// Check for changes (uncomment/comment to choose which values should be compared!)
IF ( (iVehicleID >= 1) AND (iVehicleID <= MM_MAX_NUMBER_OF_VEHICLE_ELEMENTS) ) THEN
	IF ( 	(aReadVehicleData[iVehicleID].stVehicle.bDataValid <> aOldVehicleData[iVehicleID].bDataValid) OR
			(aReadVehicleData[iVehicleID].stVehicle.bMaterial <> aOldVehicleData[iVehicleID].bMaterial) OR
			(aReadVehicleData[iVehicleID].stVehicle.bNOK <> aOldVehicleData[iVehicleID].bNOK) OR
			(aReadVehicleData[iVehicleID].stVehicle.bTool <> aOldVehicleData[iVehicleID].bTool) OR
			(aReadVehicleData[iVehicleID].stVehicle.bVehiclePresent <> aOldVehicleData[iVehicleID].bVehiclePresent) OR
//			(aReadVehicleData[iVehicleID].stVehicle.fPosition <> aOldVehicleData[iVehicleID].fPosition) OR
//			(aReadVehicleData[iVehicleID].stVehicle.fTargetPosition <> aOldVehicleData[iVehicleID].fTargetPosition) OR
//			(aReadVehicleData[iVehicleID].stVehicle.fVelocity <> aOldVehicleData[iVehicleID].fVelocity) OR
//			(aReadVehicleData[iVehicleID].stVehicle.nPathID <> aOldVehicleData[iVehicleID].nPathID) OR
			(aReadVehicleData[iVehicleID].stVehicle.nPriority <> aOldVehicleData[iVehicleID].nPriority) OR
//			(aReadVehicleData[iVehicleID].stVehicle.nState <> aOldVehicleData[iVehicleID].nState) OR
//			(aReadVehicleData[iVehicleID].stVehicle.nTargetPathID <> aOldVehicleData[iVehicleID].nTargetPathID) OR
			(aReadVehicleData[iVehicleID].stVehicle.nTicket <> aOldVehicleData[iVehicleID].nTicket) OR
			(aReadVehicleData[iVehicleID].stVehicle.nTicketSize <> aOldVehicleData[iVehicleID].nTicketSize) OR
			(aReadVehicleData[iVehicleID].stVehicle.nVehicleID <> aOldVehicleData[iVehicleID].nVehicleID) OR
			(aReadVehicleData[iVehicleID].stVehicle.sCarrierID <> aOldVehicleData[iVehicleID].sCarrierID) OR
			(aReadVehicleData[iVehicleID].stVehicle.sCurrentStationID <> aOldVehicleData[iVehicleID].sCurrentStationID) OR
			(aReadVehicleData[iVehicleID].stVehicle.sJobID <> aOldVehicleData[iVehicleID].sJobID) OR
			(aReadVehicleData[iVehicleID].stVehicle.sLastScan <> aOldVehicleData[iVehicleID].sLastScan) OR
			(aReadVehicleData[iVehicleID].stVehicle.sMaterialID <> aOldVehicleData[iVehicleID].sMaterialID) OR
			(aReadVehicleData[iVehicleID].stVehicle.sOwnerCell <> aOldVehicleData[iVehicleID].sOwnerCell) OR
			(aReadVehicleData[iVehicleID].stVehicle.sTargetStationID <> aOldVehicleData[iVehicleID].sTargetStationID) OR
			(aReadVehicleData[iVehicleID].stVehicle.sToolID <> aOldVehicleData[iVehicleID].sToolID)
		) THEN
		// Change detected. Return TRUE
		M_UpdateStatusCompare := TRUE;
		RETURN;
	END_IF
END_IF

M_UpdateStatusCompare := FALSE;
END_METHOD

METHOD PROTECTED M_VehicleIDToCarrierID : STRING(30)
VAR_INPUT
	nVehicleID		: UINT;
END_VAR

VAR
	i: INT;
END_VAR


IF (nVehicleID > 0 AND nVehicleID <= MM_MAX_NUMBER_OF_VEHICLE_ELEMENTS) THEN
	M_VehicleIDToCarrierID := aReadVehicleData[nVehicleID].stVehicle.sCarrierID;
	
ELSE
	M_VehicleIDToCarrierID := '';
	
END_IF
END_METHOD

/// Adds a vehicle to list of vehicles to read evnet-driven data from
METHOD M_VehicleToReadAdd : BOOL
VAR_INPUT
	iVehicleNo		: UINT;
END_VAR
VAR
	i				: UINT;
END_VAR

IF (iVehicleNo > 0 AND iVehicleNo <= MM_MAX_NUMBER_OF_VEHICLE_ELEMENTS) THEN
	FOR i := 1 TO MM_MAX_NUMBER_OF_VEHICLE_ELEMENTS BY 1 DO
		IF (anVehiclesToRead[i] = iVehicleNo) THEN
			// Vehicle is already added
			M_VehicleToReadAdd := TRUE;
			RETURN;
		
		ELSIF (anVehiclesToRead[i] = 0) THEN
			// Empty index found
			anVehiclesToRead[i] := iVehicleNo;
			M_VehicleToReadAdd := TRUE;
			RETURN;
			
		END_IF
	END_FOR
	
ELSE
	// Not within range
	M_VehicleToReadAdd := FALSE;
	
END_IF
END_METHOD

/// Removes a vehicle from list of vehicles to read evnet-driven data from
METHOD M_VehicleToReadRemove : BOOL
VAR_INPUT
	iVehicleNo		: UINT;
END_VAR
VAR
	i				: UINT;
END_VAR

IF (iVehicleNo > 0 AND iVehicleNo <= MM_MAX_NUMBER_OF_VEHICLE_ELEMENTS) THEN
	FOR i := 1 TO MM_MAX_NUMBER_OF_VEHICLE_ELEMENTS BY 1 DO
		IF (anVehiclesToRead[i] = iVehicleNo) THEN
			// Vehicle is found
			anVehiclesToRead[i] := 0;
			M_VehicleToReadRemove := TRUE;
			RETURN;
			
		END_IF
	END_FOR
	
ELSE
	// Not within range
	M_VehicleToReadRemove := FALSE;
	
END_IF
END_METHOD

PROPERTY PUBLIC P_bForceVehicleUpdateOPC : BOOL
GET
P_bForceVehicleUpdateOPC := bForceVehicleUpdateOPC;
END_GET
SET
bForceVehicleUpdateOPC := P_bForceVehicleUpdateOPC;
END_SET
END_PROPERTY

/// When TRUE it is OK to run DecisionPoint, ExitPoint and Buffer handling
PROPERTY PUBLIC P_bTrackReady : BOOL
GET
// TRUE if track client is ready to use
P_bTrackReady := bEnable AND bConnectedMethod AND bConnectedNode AND bTrackInitDone AND (eTrackState = E_TrackState.Started);
END_GET
END_PROPERTY

PROPERTY PUBLIC P_eCellType : E_CellType
GET
P_eCellType := eCellType;
END_GET
SET
eCellType := P_eCellType;
END_SET
END_PROPERTY

PROPERTY PUBLIC P_nTrackserverPort : UINT
GET
P_nTrackserverPort := nTrackServerPortNo;
END_GET
SET
nTrackServerPortNo := P_nTrackserverPort;
END_SET
END_PROPERTY

PROPERTY PUBLIC P_rErrorResetDelay : REAL
GET
P_rErrorResetDelay := rErrorResetDelay;
END_GET
SET
rErrorResetDelay := P_rErrorResetDelay;
END_SET
END_PROPERTY

PROPERTY PUBLIC P_rPollingInterval : REAL
GET
P_rPollingInterval := rReadInterval;
END_GET
SET
rReadInterval := P_rPollingInterval;
END_SET
END_PROPERTY

PROPERTY PUBLIC P_sCellID : STRING(30)
GET
P_sCellID := sCellID;
END_GET
SET
sCellID := F_ToUCase(P_sCellID);
END_SET
END_PROPERTY

PROPERTY PUBLIC P_sNextStationOnTrack : STRING(30)
GET
P_sNextStationOnTrack := sNextStationOnTrack;
END_GET
SET

IF (LEN(P_sNextStationOnTrack) > 0) THEN
	sNextStationOnTrack := P_sNextStationOnTrack;
END_IF
END_SET
END_PROPERTY

PROPERTY PUBLIC P_sTrackserverNetID : STRING
GET
P_sTrackserverNetID := sTrackServerNetID;
END_GET
SET
sTrackServerNetID := P_sTrackserverNetID;
END_SET
END_PROPERTY

PROPERTY PUBLIC P_sTrackserverURL : STRING
GET
P_sTrackserverURL := sTrackServerUrl;
END_GET
SET
sTrackServerUrl := P_sTrackserverURL;
END_SET
END_PROPERTY

END_FUNCTION_BLOCK

// ---- ECC/Basic/ADS Comm/FB_ADS_Comm.TcPOU
FUNCTION_BLOCK FB_ADS_Comm
VAR_INPUT
	bEnable				: BOOL;			// TRUE to run communication
	eType				: E_ADS_Comm_Type;// Read or write
	rInterval			: REAL;			// Update interval [s]
	pLocalVar			: PVOID;		// Pointer to local variable to link to remote device
	nLocalSize			: UINT;			// Size of local variable
	sNetID				: T_AmsNetId;	// ADS address on remote ADS device
	nPort				: T_AmsPort;	// ADS port on remote ADS device
	sVarName			: STRING;		// Remote symbol name to read/write
END_VAR
VAR_OUTPUT
	bWriteError			: BOOL;			// Writing error
	bReadError			: BOOL;			// Reading error
	bParameterError		: BOOL;			// Parameter error
END_VAR
VAR
	fbReadAds			: FB_ReadAdsSymByName;	// FB to read symbols via. ADS
	fbWriteAds 			: FB_WriteAdsSymByName;	// FB to write symbols via. ADS
	nState				: E_ADS_Comm_State;		// State
	tonExecute			: TON;					// Execute timer
	tonInterval			: TON;					// For calculating actual read/write interval
	rActInterval		: REAL;					// [s] Measured read/write interval
	bSendRecv			: BOOL;					// TRUE to read or write data
	bSendRecvDone		: BOOL;					// TRUE when completed
END_VAR

IF (bEnable) THEN
	// Check parameters
	IF (sNetID = '') THEN
		bParameterError := TRUE;
	ELSIF (nPort = 0) THEN
		bParameterError := TRUE;
	ELSIF (pLocalVar = 0) THEN
		bParameterError := TRUE;
	ELSIF (nLocalSize <= 0) THEN
		bParameterError := TRUE;
	ELSE
		bParameterError := FALSE;
	END_IF
ELSE
	bParameterError := FALSE;
	bReadError := FALSE;
	bWriteError := FALSE;
	bSendRecvDone := FALSE;
END_IF

// Check interval
IF (rInterval < 0) THEN
	rInterval := 0;
END_IF

// Run read FB
IF (bEnable) THEN
	// ADS communication
	CASE nState OF
		E_ADS_Comm_State.Disabled:
			bWriteError := FALSE;
			bReadError := FALSE;
			bParameterError := FALSE;
			tonExecute.IN := FALSE;
			fbReadAds.bRead := FALSE;
			fbWriteAds.bWrite := FALSE;
			IF (bEnable) THEN
				nState := E_ADS_Comm_State.Idle;
			END_IF

		E_ADS_Comm_State.Idle:
			tonExecute.IN := TRUE;
			IF (NOT bEnable) THEN
				nState := E_ADS_Comm_State.Disabled;
			ELSIF (eType = ADS_RD_FAST) THEN
				nState := E_ADS_Comm_State.Wait_Read;
			ELSIF (eType = ADS_WR_FAST) THEN
				nState := E_ADS_Comm_State.Wait_Write;
			ELSIF (eType = ADS_RD_SLOW) THEN
				nState := E_ADS_Comm_State.Wait_Read;
			ELSIF (eType = ADS_WR_SLOW) THEN
				nState := E_ADS_Comm_State.Wait_Write;
			ELSIF (eType = ADS_WR_TRIG1) THEN
				nState := E_ADS_Comm_State.Wait_Write;
			ELSIF (eType = ADS_WR_TRIG2) THEN
				nState := E_ADS_Comm_State.Wait_Write;
			ELSIF (eType = ADS_WR_TRIG3) THEN
				nState := E_ADS_Comm_State.Wait_Write;
			END_IF

		E_ADS_Comm_State.Wait_Write:
			IF (tonExecute.Q OR bSendRecv) THEN
				tonExecute.IN := FALSE;
				fbWriteAds.bWrite := TRUE;
				fbWriteAds.sNetID := sNetID; 
				fbWriteAds.nPort := nPort; 
				fbWriteAds.sVarName := sVarName; 
				fbWriteAds.nSrcAddr := pLocalVar;
				fbWriteAds.nLen := nLocalSize;
//				fbWriteAds.eComMode := eAdsComModeFastCom;
				fbWriteAds.eComMode := eAdsComModeSecureCom;
				nState := E_ADS_Comm_State.Writing;		
			END_IF

		E_ADS_Comm_State.Writing:
			IF (fbWriteAds.bBusy) THEN
				tonExecute.IN := TRUE;
			ELSE
				fbWriteAds.bWrite := FALSE;
				IF (fbWriteAds.bError) THEN
					nState := E_ADS_Comm_State.Write_Error;
				ELSE
					rActInterval := (TIME_TO_REAL(tonInterval.ET) / 1000.0);
					tonInterval(IN := FALSE);
					bWriteError := FALSE;
					bSendRecvDone := TRUE;
					nState := E_ADS_Comm_State.Idle;
				END_IF
			END_IF

		E_ADS_Comm_State.Write_Error:
			bWriteError := TRUE;		
			nState := E_ADS_Comm_State.Idle;

		E_ADS_Comm_State.Wait_Read:
			IF (tonExecute.Q OR bSendRecv) THEN
				tonExecute.IN := FALSE;
				fbReadAds.bRead := TRUE;
				fbReadAds.sNetID := sNetID;
				fbReadAds.nPort := nPort; 
				fbReadAds.sVarName := sVarName; 
				fbReadAds.nDestAddr := pLocalVar;
				fbReadAds.nLen := nLocalSize;
//				fbReadAds.eComMode := eAdsComModeFastCom;
				fbReadAds.eComMode := eAdsComModeSecureCom;
				nState := E_ADS_Comm_State.Reading;	
			END_IF

		E_ADS_Comm_State.Reading:
			IF (fbReadAds.bBusy) THEN
				tonExecute.IN := TRUE;
			ELSE
				fbReadAds.bRead := FALSE;
				IF (fbReadAds.bError) THEN
					nState := E_ADS_Comm_State.Read_Error;
				ELSE
					rActInterval := (TIME_TO_REAL(tonInterval.ET) / 1000.0);
					tonInterval(IN := FALSE);
					bReadError := FALSE;
					bSendRecvDone := TRUE;
					nState := E_ADS_Comm_State.Idle;
				END_IF
			END_IF
		
		E_ADS_Comm_State.Read_Error:
			bReadError := TRUE;		
			nState := E_ADS_Comm_State.Idle;

		ELSE
			nState := E_ADS_Comm_State.Disabled;
	END_CASE

	IF ((eType = ADS_WR_TRIG1) OR (eType = ADS_WR_TRIG2) OR (eType = ADS_WR_TRIG3) OR
		(eType = ADS_RD_TRIG1) OR (eType = ADS_RD_TRIG2) OR (eType = ADS_RD_TRIG3)) THEN
		// No cyclic reading/writing
		tonExecute.IN := FALSE;
	END_IF
	tonExecute.PT := REAL_TO_TIME(rInterval * 1000.0);
	tonExecute();
	tonInterval(IN := TRUE, PT := T#60S);
	fbReadAds.tTimeout := DEFAULT_ADS_TIMEOUT;
	fbReadAds();
	fbWriteAds();
	fbWriteAds.tTimeout := DEFAULT_ADS_TIMEOUT;

END_IF

METHOD PUBLIC M_SendRecv : BOOL
VAR_INPUT
END_VAR
IF ((eType = E_ADS_Comm_Type.ADS_WR_TRIG1) OR (eType = E_ADS_Comm_Type.ADS_RD_TRIG1) OR
	(eType = E_ADS_Comm_Type.ADS_WR_TRIG2) OR (eType = E_ADS_Comm_Type.ADS_RD_TRIG2) OR
	(eType = E_ADS_Comm_Type.ADS_WR_TRIG3) OR (eType = E_ADS_Comm_Type.ADS_RD_TRIG3)) THEN
	
	IF (NOT bSendRecv) THEN
		bSendRecvDone := FALSE;	
	END_IF
	bSendRecv := TRUE;
END_IF
END_METHOD

METHOD PUBLIC M_SendRecvCompleted : BOOL
VAR_INPUT
END_VAR
M_SendRecvCompleted := bSendRecvDone;
END_METHOD

METHOD PUBLIC M_SendRecvStop : BOOL
VAR_INPUT
END_VAR
bSendRecv := FALSE;
END_METHOD

END_FUNCTION_BLOCK

// ---- ECC/TrackClient/Station Control/FB_StationControl.TcPOU
FUNCTION_BLOCK FB_StationControl
VAR_IN_OUT
	stStationData			: ST_MMStation;
END_VAR
VAR_INPUT
// From station FB
	bReadyForVehicleInput	: BOOL;		// TRUE when station is ready for a vehicle/last at input location
	bCompletedInput			: BOOL;		// TRUE when part operation has finished (ready to deliver to vehicle on input)
	bReadyForVehicleOutput	: BOOL;		// TRUE when station is ready for a vehicle/last at output location
	bCompletedOutput		: BOOL;		// TRUE when part operation has finished (ready to deliver to vehicle on input)
// From Track Client FB (Vehicle movement)
	bVehiclePreMoved		: BOOL;
	bVehiclePostMoved		: BOOL;
	bVehiclePreToInMoved	: BOOL;
	bVehiclePreToOutMoved	: BOOL;
	bVehicleInToOutMoved	: BOOL;
	bVehicleInToPostMoved	: BOOL;
	bVehicleOutToPostMoved	: BOOL;
END_VAR
VAR_OUTPUT
// To Station FB
	bVehicleReadyAtInput	: BOOL;		// Set to TRUE when a vehicle is ready at the station input location
	bVehicleReadyAtOutput	: BOOL;		// Set to TRUE when a vehicle is ready at the station input location
// To Track Client (vehicle movement)
	bMoveVehiclePreToIn		: BOOL;		// TRUE when a vehicle need to be moved from pre buffer to station input/1 location
	bMoveVehiclePreToOut	: BOOL;		// TRUE when a vehicle need to be moved from pre buffer to station output/2 location
	bMoveVehicleInToOut		: BOOL;		// TRUE when a vehicle need to be moved from station input/1 to station output/2
	bMoveVehicleInToPost	: BOOL;		// TRUE when a vehicle need to be moved from station input/1 to post buffer
	bMoveVehicleOutToPost	: BOOL;		// TRUE when a vehicle need to be moved from station output/2 to post buffer
END_VAR
VAR
	bInitDone				: BOOL;	

	// In to station
	eStationInState			: E_StationInOutState;
	
	// Out from station
	eStationOutState		: E_StationInOutState;
	
	// Misc
	i						: UINT;
	
	// TEST
	bTEST_ForceCompletedInput	: BOOL;
	bTEST_ForceCompletedOutput	: BOOL;
END_VAR
VAR CONSTANT
	
END_VAR


// Init
M_Init();

// Buffer handling... Decide which vehicles to move in the buffers
//M_Buffers();

// Station handling
M_Station();

METHOD PUBLIC M_AddVehicle : USINT
VAR_INPUT
	nTicket			: UINT;
	nVehicleID		: UINT;
	nPriority		: UINT;
END_VAR
VAR
	i				: USINT;
	iFoundIndex		: USINT;
END_VAR
// Return TRUE if station is ready to receive the specified task/ticket/priority

iFoundIndex := 0;

// Find the empty spot closest to station position (smallest index)
FOR i := iPreBufferSize TO 1 BY -1 DO
	IF (stStationData.astPreBuffer[i].nCurrentVehicleID = 0) THEN
		// Buffer spot is empty
		iFoundIndex := i;
	ELSE
		EXIT;
	END_IF
END_FOR

IF (iFoundIndex > 0) THEN
	stStationData.astPreBuffer[iFoundIndex].nReservedVehicleID := nVehicleID;
	stStationData.astPreBuffer[iFoundIndex].nTicket := nTicket;
	stStationData.astPreBuffer[iFoundIndex].CurrentPriority := nPriority;
	stStationData.astPreBuffer[iFoundIndex].nCurrentVehicleID := nVehicleID;
END_IF

M_AddVehicle := iFoundIndex;
END_METHOD

/// Handling of the pre/post buffer on the station
METHOD M_Buffers
VAR_INPUT
END_VAR

/////////////////////////////////////////////////////////////////////////////////////////////////////////////////////////////////////////////////////////
// Pre buffer
/////////////////////////////////////////////////////////////////////////////////////////////////////////////////////////////////////////////////////////		
CASE ePreBufferState OF
	E_StationBufferState.Idle:
		bMoveVehiclePre := FALSE;
		iBufferSourcePre := 0;
		iBufferTargetPre := 0;
		iPreBufferIdx := 0;

	E_StationBufferState.CheckBuffer:
		iPreBufferIdx := iPreBufferIdx + 1;
		IF (iPreBufferIdx < MM_MAX_BUFFER_INDEX) THEN
			IF ( (stStationData.astPreBuffer[iPreBufferIdx].nCurrentVehicleID = 0) AND (stStationData.astPreBuffer[iPreBufferIdx].bPresent) ) THEN
				// Buffer space empty... Check next index
				IF ( (stStationData.astPreBuffer[iPreBufferIdx+1].nCurrentVehicleID > 0) AND (stStationData.astPreBuffer[iPreBufferIdx+1].bPresent) ) THEN
					// Buffer occupied, move to previous buffer index (closer to station pickup position)
					ePreBufferState := E_StationBufferState.StartMove;
				END_IF
			END_IF
		ELSE
			// All buffer indexes checked
			ePreBufferState := E_BufferState.Idle;
		END_IF
		
	E_StationBufferState.StartMove:
		bMoveVehiclePre := TRUE;
		iBufferSourcePre := iPreBufferIdx+1;
		iBufferTargetPre := iPreBufferIdx;
		ePreBufferState := E_StationBufferState.WaitMove;
		
	E_StationBufferState.WaitMove:
		IF (bVehiclePreMoved) THEN
			bMoveVehiclePre := FALSE;
			ePreBufferState := E_BufferState.Idle;			
		END_IF

END_CASE


/////////////////////////////////////////////////////////////////////////////////////////////////////////////////////////////////////////////////////////
// Post buffer
/////////////////////////////////////////////////////////////////////////////////////////////////////////////////////////////////////////////////////////		
CASE ePostBufferState OF
	E_StationBufferState.Idle:
		bMoveVehiclePost := FALSE;
		iBufferSourcePost := 0;
		iBufferTargetPost := 0;
		iPostBufferIdx := MM_MAX_BUFFER_INDEX+1;

	E_StationBufferState.CheckBuffer:
		iPostBufferIdx := iPostBufferIdx - 1;
		IF (iPostBufferIdx > 1) THEN
			IF ( (stStationData.astPostBuffer[iPostBufferIdx].nCurrentVehicleID = 0) AND (stStationData.astPostBuffer[iPostBufferIdx].bPresent) ) THEN
				// Buffer space empty... Check next index
				IF ( (stStationData.astPostBuffer[iPostBufferIdx-1].nCurrentVehicleID > 0) AND (stStationData.astPostBuffer[iPostBufferIdx-1].bPresent) ) THEN
					// Buffer occupied, move to next buffer index (closer to exit point)
					ePostBufferState := E_StationBufferState.StartMove;
				END_IF
			END_IF
		ELSE
			// All buffer indexes checked
			ePostBufferState := E_BufferState.Idle;
		END_IF
		
	E_StationBufferState.StartMove:
		bMoveVehiclePost := TRUE;
		iBufferSourcePost := iPostBufferIdx-1;
		iBufferTargetPost := iPostBufferIdx;
		ePostBufferState := E_StationBufferState.WaitMove;
		
	E_StationBufferState.WaitMove:
		IF (bVehiclePostMoved) THEN
			bMoveVehiclePost := FALSE;
			ePostBufferState := E_BufferState.Idle;			
		END_IF

END_CASE
END_METHOD

METHOD M_ClearAll : BOOL
VAR_INPUT
END_VAR
bVehicleReadyAtInput := FALSE;
bVehicleReadyAtOutput := FALSE;
bMoveVehiclePreToIn := FALSE;
bMoveVehiclePreToOut := FALSE;
bMoveVehicleInToOut	 := FALSE;
bMoveVehicleInToPost := FALSE;
bMoveVehicleOutToPost := FALSE;

eStationInState	:= E_StationInOutState.Idle;
eStationOutState := E_StationInOutState.Idle;


F_Logfile('StationControl - All data cleared!');

M_ClearAll:= TRUE;
END_METHOD

METHOD PUBLIC M_Init
VAR_INPUT
END_VAR
VAR
	i		: UINT;
END_VAR
// Init all variables (deletes values!)
IF (NOT bInitDone) THEN
	bInitDone := TRUE;
END_IF
END_METHOD

METHOD PUBLIC M_PostBufferEmpty : BOOL
VAR_INPUT
END_VAR
// Returns TRUE if post-buffer is empty
M_PostBufferEmpty := iPostBufferFree >= iPostBufferSize;
END_METHOD

METHOD PUBLIC M_PreBufferEmpty : BOOL
VAR_INPUT
END_VAR
// Returns TRUE if pre-buffer is empty
M_PreBufferEmpty := iPreBufferFree >= iPreBufferSize;
END_METHOD

METHOD PUBLIC M_RemoveVehicle : UINT
VAR_INPUT
	nCarrierID		: UINT;
END_VAR
VAR
	i				: UINT;
END_VAR

// Find the empty spot closes to station position (smallest index)
FOR i := iPostBufferSize TO 1 BY -1 DO
	IF (stStationData.astPostBuffer[i].nCurrentVehicleID = nCarrierID) THEN
		MEMSET(ADR(stStationData.astPostBuffer[i]), 0, SIZEOF(stStationData.astPostBuffer[i]));
		M_RemoveVehicle := i;
		RETURN;
	END_IF
END_FOR

M_RemoveVehicle := 0;
END_METHOD

METHOD PUBLIC M_ShiftForward : BOOL
VAR_INPUT
END_VAR
VAR
	i		: UINT;
END_VAR
// Shift buffer spaces (move all items one spot forward)

// Post buffer shift
FOR i := MM_MAX_BUFFER_INDEX TO 1 BY -1 DO
	IF (stStationData.astPostBuffer[i].bPresent) THEN
		stStationData.astPostBuffer[i].nReservedVehicleID := stStationData.astPostBuffer[i-1].nReservedVehicleID;
		stStationData.astPostBuffer[i].nCurrentVehicleID := stStationData.astPostBuffer[i-1].nCurrentVehicleID;
		stStationData.astPostBuffer[i].nTicket := stStationData.astPostBuffer[i-1].nTicket;
		stStationData.astPostBuffer[i].CurrentPriority := stStationData.astPostBuffer[i-1].CurrentPriority;
	END_IF
END_FOR

// Station data to post buffer
stStationData.astPostBuffer[1] := stStationData.stStationData;

// Pre buffer last space to station data
stStationData.stStationData := stStationData.astPreBuffer[1];

// Pre buffer shift
FOR i := 1 TO MM_MAX_BUFFER_INDEX-1 BY 1 DO
	IF (stStationData.astPreBuffer[i].bPresent) THEN
		stStationData.astPreBuffer[i].nReservedVehicleID := stStationData.astPreBuffer[i+1].nReservedVehicleID;
		stStationData.astPreBuffer[i].nCurrentVehicleID := stStationData.astPreBuffer[i+1].nCurrentVehicleID;
		stStationData.astPreBuffer[i].nTicket := stStationData.astPreBuffer[i+1].nTicket;
		stStationData.astPreBuffer[i].CurrentPriority := stStationData.astPreBuffer[i+1].CurrentPriority;
	END_IF
END_FOR
END_METHOD

METHOD PROTECTED M_Station
VAR_INPUT
END_VAR

/////////////////////////////////////////////////////////////////////////////////////////////////////////////////////////////////////////////////////////
// Into station
/////////////////////////////////////////////////////////////////////////////////////////////////////////////////////////////////////////////////////////		
CASE eStationInState OF
	E_StationInOutState.Idle:
		bMoveVehiclePreToOut := FALSE;
		bMoveVehiclePreToIn := FALSE;
		eStationInState := E_StationInOutState.Check;
		
	E_StationInOutState.Check:
		IF (bReadyForVehicleInput AND (stStationData.stStationData1.nCurrentVehicleID = 0) ) THEN
			// Station input location is ready for a vehicle
			IF (stStationData.astPreBuffer[1].nCurrentVehicleID > 0) THEN
				// Vehicle is ready in pre buffer location closest to station
				eStationInState := E_StationInOutState.StartMoveIn;
			END_IF
		ELSIF (bReadyForVehicleOutput AND (stStationData.stStationData2.nCurrentVehicleID = 0) ) THEN
			// Station output location is ready for a vehicle
			IF (stStationData.astPreBuffer[1].nCurrentVehicleID > 0) THEN
				// Vehicle is ready in pre buffer location closest to station
				eStationInState := E_StationInOutState.StartMoveOut;
			END_IF			
		END_IF
	
	E_StationInOutState.StartMoveOut:
		bMoveVehiclePreToOut := TRUE;
		F_LogLine('TC_STAT Move to Out: %d', stStationData.astPreBuffer[1].nCurrentVehicleID);
		eStationInState := E_StationInOutState.WaitMoveOut;
	
	E_StationInOutState.WaitMoveOut:
		IF (bVehiclePreToOutMoved) THEN
			bMoveVehiclePreToOut := FALSE;
			bVehicleReadyAtOutput := TRUE;
			F_LogLine('TC_STAT Move to Out Done! ', 0);
			eStationInState := E_StationInOutState.Idle;
		END_IF

	E_StationInOutState.StartMoveIn:
		bMoveVehiclePreToIn := TRUE;
		F_LogLine('TC_STAT Move to In: %d', stStationData.astPreBuffer[1].nCurrentVehicleID);
		eStationInState := E_StationInOutState.WaitMoveIn;
	
	E_StationInOutState.WaitMoveIn:
		IF (bVehiclePreToInMoved) THEN
			bMoveVehiclePreToIn := FALSE;
			bVehicleReadyAtInput := TRUE;
			F_LogLine('TC_STAT Move to In Done! ', 0);
			eStationInState := E_StationInOutState.Idle;
		END_IF
	
	ELSE
		eStationInState := E_StationInOutState.Idle;
		
END_CASE



/////////////////////////////////////////////////////////////////////////////////////////////////////////////////////////////////////////////////////////
// Out from station
/////////////////////////////////////////////////////////////////////////////////////////////////////////////////////////////////////////////////////////		
CASE eStationOutState OF
	E_StationInOutState.Idle:
		bMoveVehicleInToPost := FALSE;
		bMoveVehicleOutToPost := FALSE;
		eStationOutState := E_StationInOutState.Check;
		
	E_StationInOutState.Check:
		IF ((bCompletedInput OR bTEST_ForceCompletedInput) AND (stStationData.stStationData1.nCurrentVehicleID > 0) ) THEN
			// Station input location is completed and has a vehicle
			bTEST_ForceCompletedInput := FALSE;
			IF (stStationData.astPostBuffer[1].nCurrentVehicleID = 0) THEN
				// No vehicle in post buffer location closest to station
				eStationOutState := E_StationInOutState.StartMoveIn;
			END_IF
		ELSIF ((bCompletedOutput OR bTEST_ForceCompletedOutput) AND (stStationData.stStationData2.nCurrentVehicleID > 0) ) THEN
			// Station output location is ready for a vehicle
			bTEST_ForceCompletedOutput := FALSE;
			IF (stStationData.astPostBuffer[1].nCurrentVehicleID = 0) THEN
				// No vehicle in post buffer location closest to station
				eStationOutState := E_StationInOutState.StartMoveOut;
			END_IF			
		END_IF
	
	E_StationInOutState.StartMoveOut:
		bMoveVehicleOutToPost := TRUE;
		bVehicleReadyAtOutput := FALSE;
		F_LogLine('TC_STAT Move from Out: %d', stStationData.stStationData2.nCurrentVehicleID);
		eStationOutState := E_StationInOutState.WaitMoveOut;
	
	E_StationInOutState.WaitMoveOut:
		IF (bVehicleOutToPostMoved) THEN
			bMoveVehicleOutToPost := FALSE;
			F_LogLine('TC_STAT Move from Out Done! ', 0);
			eStationOutState := E_StationInOutState.Idle;
		END_IF

	E_StationInOutState.StartMoveIn:
		bMoveVehicleInToPost := TRUE;
		bVehicleReadyAtInput := FALSE;
		F_LogLine('TC_STAT Move from In: %d', stStationData.stStationData1.nCurrentVehicleID);
		eStationOutState := E_StationInOutState.WaitMoveIn;
	
	E_StationInOutState.WaitMoveIn:
		IF (bVehicleInToPostMoved) THEN
			bMoveVehicleInToPost := FALSE;
			F_LogLine('TC_STAT Move from In Done! ', 0);
			eStationOutState := E_StationInOutState.Idle;
		END_IF
	
	ELSE
		eStationOutState := E_StationInOutState.Idle;
		
END_CASE
END_METHOD

PROPERTY PUBLIC P_bPresent : BOOL
GET
P_bPresent := stStationData.bPresent;
END_GET
SET
stStationData.bPresent := P_bPresent;
END_SET
END_PROPERTY

PROPERTY PUBLIC P_bReInit : BOOL
SET
bInitDone := P_bReInit;
END_SET
END_PROPERTY

/// NOTE; Only needed because VehicleReadyAtInput is set from decision point logic and not from inside StationControl FB
PROPERTY PUBLIC P_bVehicleReadyAtInput : BOOL
GET
P_bVehicleReadyAtInput := bVehicleReadyAtInput;
END_GET
SET
bVehicleReadyAtInput := P_bVehicleReadyAtInput;
END_SET
END_PROPERTY

PROPERTY PUBLIC P_sCellID : STRING(30)
GET
P_sCellID := stStationData.sCellID;
END_GET
SET
stStationData.sCellID := P_sCellID;
END_SET
END_PROPERTY

PROPERTY PUBLIC P_sStationID : STRING(30)
GET
P_sStationID := stStationData.sStationID;
END_GET
SET
stStationData.sStationID := P_sStationID;
END_SET
END_PROPERTY

END_FUNCTION_BLOCK

// ---- ECC/TrackClient/Buffer Control/FB_BufferControl.TcPOU
/// Controls pre-buffer and post-buffer on stations
FUNCTION_BLOCK FB_BufferControl
VAR_IN_OUT
	stMMBuffer : ARRAY[1..MM_MAX_BUFFER_INDEX] OF ST_MMBuffer;
END_VAR
VAR_INPUT
END_VAR
VAR_OUTPUT
END_VAR
VAR
	iBufferSize			: UINT := MM_MAX_BUFFER_INDEX;
	sBufferType			: STRING(4); //Pre / Post
	aBufferCmdID 		: ARRAY [1..MM_MAX_BUFFER_INDEX] OF UINT;
END_VAR

/// Adds a new vehicle to the buffer, taking up an additional space in the buffer
/// Returns FALSE if not able to add the vehicle!
METHOD PUBLIC M_AddVehicle : BOOL
VAR_INPUT
	iVehicleID			: UINT;
	iTicket				: UINT;
	iTicketSize			: UINT;
	iPriority			: UINT;
	iMoveCmdID			: UINT;
END_VAR
VAR
	i					: UINT;
END_VAR

IF ( (iVehicleID > 0) AND (iMoveCmdID > 0) AND (sBufferType = 'Pre' OR sBufferType = 'Post' ) ) THEN
	// Find first empty space in buffer
	IF sBufferType = 'Pre' THEN
		FOR i := 1 TO (iBufferSize) BY 1 DO
			IF (aBufferCmdID[i] = 0) THEN
				aBufferCmdID[i] := iMoveCmdID;
	
				stMMBuffer[i].nReservedVehicleID := iVehicleID;
				stMMBuffer[i].nCurrentVehicleID := iVehicleID;
				stMMBuffer[i].nTicket := iTicket;
				stMMBuffer[i].nTicketSize := iTicketSize;
				stMMBuffer[i].CurrentPriority := iPriority;						
				
				M_AddVehicle := TRUE;
				
				F_LogLine('TC_BUFCTRL: Vehicle added in Pre buffer : %d', iVehicleID);
				RETURN;
				
			END_IF
		END_FOR
	ELSIF sBufferType = 'Post' THEN
		FOR i := (iBufferSize) TO 1 BY -1 DO
			IF (aBufferCmdID[i] = 0) THEN
				aBufferCmdID[i] := iMoveCmdID;
	
				stMMBuffer[i].nReservedVehicleID := iVehicleID;
				stMMBuffer[i].nCurrentVehicleID := iVehicleID;
				stMMBuffer[i].nTicket := iTicket;
				stMMBuffer[i].nTicketSize := iTicketSize;
				stMMBuffer[i].CurrentPriority := iPriority;						
				
				M_AddVehicle := TRUE;
				
				F_LogLine('TC_BUFCTRL: Vehicle added in Post buffer : %d', iVehicleID);
				RETURN;
				
			END_IF
		END_FOR
	END_IF	
ELSE
	// No vehicle to remove
	M_AddVehicle := FALSE;
	RETURN;
	
END_IF
END_METHOD

METHOD M_ClearAll : BOOL
VAR_INPUT
END_VAR
VAR
	i	: UINT;
END_VAR

FOR i:=1 TO MM_MAX_BUFFER_INDEX DO
	IF stMMBuffer[i].bPresent THEN
		stMMBuffer[i].CurrentPriority := 0;
		stMMBuffer[i].nCurrentVehicleID := 0;
		stMMBuffer[i].nReservedVehicleID := 0;
		stMMBuffer[i].nTicket := 0;
		stMMBuffer[i].nTicketSize := 0;
		aBufferCmdID[i] := 0;
	END_IF
END_FOR
	
F_Logfile('BFCtrl - All data cleared!');

M_ClearAll := TRUE;
END_METHOD

METHOD PUBLIC M_IsEmpty : BOOL
VAR_INPUT
END_VAR

IF (sBufferType = 'Pre' AND (stMMBuffer[1].nCurrentVehicleID = 0)) OR (sBufferType = 'Post' AND ( stMMBuffer[iBufferSize].nCurrentVehicleID = 0))THEN
	M_IsEmpty := TRUE;
	
ELSE
	M_IsEmpty := FALSE;
	
END_IF
END_METHOD

METHOD PUBLIC M_IsFull : BOOL
VAR_INPUT
END_VAR

IF (sBufferType = 'Pre' AND (stMMBuffer[iBufferSize].nCurrentVehicleID > 0)) OR (sBufferType = 'Post' AND ( stMMBuffer[1].nCurrentVehicleID > 0))THEN
	M_IsFull := TRUE;
	
ELSE
	M_IsFull := FALSE;
	
END_IF
END_METHOD

/// Removes a vehicle from the buffer, freeing up one space in the buffer
/// Returns the vehicle ID of the removed vehicle (0 if not able to remove the vehicle (if buffer is empty) )
METHOD PUBLIC M_RemoveVehicle : UINT
VAR_INPUT
	iVehicleID			: UINT;
//	iTicket				: UINT;
//	iTicketSize			: UINT;
//	iPriority			: UINT;
//	iMoveCmdID			: UINT;
END_VAR
VAR
	i					: UINT;
END_VAR

IF (stMMBuffer[1].nCurrentVehicleID > 0 AND sBufferType = 'Pre') OR (stMMBuffer[iBufferSize].nCurrentVehicleID > 0 AND sBufferType = 'Post') THEN
	
	IF sBufferType = 'Pre' THEN
		// Save ID of vehicle to remove
		M_RemoveVehicle := stMMBuffer[1].nCurrentVehicleID;
		
		// Re-arrange values in array
		FOR i := 1 TO (MM_MAX_BUFFER_INDEX - 1) BY 1 DO
			stMMBuffer[i].CurrentPriority := stMMBuffer[i+1].CurrentPriority;
			stMMBuffer[i].nCurrentVehicleID := stMMBuffer[i+1].nCurrentVehicleID;
			stMMBuffer[i].nReservedVehicleID := stMMBuffer[i+1].nReservedVehicleID;
			stMMBuffer[i].nTicket := stMMBuffer[i+1].nTicket;
			stMMBuffer[i].nTicketSize := stMMBuffer[i+1].nTicketSize;
			stMMBuffer[i].stLocation := stMMBuffer[i+1].stLocation;
			aBufferCmdID[i] := aBufferCmdID[i+1];
		END_FOR
		
		F_LogLine('TC_BUFCTRL: Vehicle removed from Pre buffer : %d', M_RemoveVehicle);
	ELSIF sBufferType = 'Post' THEN
		// Save ID of vehicle to remove
		M_RemoveVehicle := stMMBuffer[iBufferSize].nCurrentVehicleID;
		
		// Re-arrange values in array
		FOR i := iBufferSize TO 2 BY -1 DO
			stMMBuffer[i] := stMMBuffer[i-1];
			aBufferCmdID[i] := aBufferCmdID[i-1];
		END_FOR
		stMMBuffer[1].CurrentPriority := stMMBuffer[MM_MAX_BUFFER_INDEX].CurrentPriority;
		stMMBuffer[1].nCurrentVehicleID := stMMBuffer[MM_MAX_BUFFER_INDEX].nCurrentVehicleID;
		stMMBuffer[1].nReservedVehicleID := stMMBuffer[MM_MAX_BUFFER_INDEX].nReservedVehicleID;
		stMMBuffer[1].nTicket := stMMBuffer[MM_MAX_BUFFER_INDEX].nTicket;
		stMMBuffer[1].nTicketSize := stMMBuffer[MM_MAX_BUFFER_INDEX].nTicketSize;
		stMMBuffer[1].stLocation := stMMBuffer[MM_MAX_BUFFER_INDEX].stLocation;
		aBufferCmdID[1] := aBufferCmdID[MM_MAX_BUFFER_INDEX];
		
		F_LogLine('TC_BUFCTRL: Vehicle removed from Post buffer : %d', M_RemoveVehicle);
	END_IF
ELSE
	// No vehicle to remove
	M_RemoveVehicle := 0;
	
END_IF
END_METHOD

/// Sets/gets buffer size. Size is limited to MM_MAX_BUFFER_INDEX
PROPERTY PUBLIC P_iBufferSize : UINT
GET
P_iBufferSize := iBufferSize;
END_GET
SET

iBufferSize := LIMIT(0, P_iBufferSize, MM_MAX_BUFFER_INDEX);
END_SET
END_PROPERTY

PROPERTY P_iCurrentVehicleCmdID : UINT
GET
IF sBufferType = 'Pre' THEN
	P_iCurrentVehicleCmdID := aBufferCmdID[1];
ELSIF sBufferType = 'Post' THEN
	P_iCurrentVehicleCmdID := aBufferCmdID[iBufferSize];
ELSE
	P_iCurrentVehicleCmdID := 0;
END_IF
END_GET
END_PROPERTY

PROPERTY P_iCurrentVehicleID : UINT
GET
IF sBufferType = 'Pre' THEN
	P_iCurrentVehicleID := stMMBuffer[1].nCurrentVehicleID;
ELSIF sBufferType = 'Post' THEN
	P_iCurrentVehicleID := stMMBuffer[iBufferSize].nCurrentVehicleID;
ELSE
	P_iCurrentVehicleID := 0;
END_IF
END_GET
END_PROPERTY

PROPERTY P_iCurrentVehicleTicket : UINT
GET
IF sBufferType = 'Pre' THEN
	P_iCurrentVehicleTicket := stMMBuffer[1].nTicket;
ELSIF sBufferType = 'Post' THEN
	P_iCurrentVehicleTicket := stMMBuffer[iBufferSize].nTicket;
ELSE
	P_iCurrentVehicleTicket := 0;
END_IF
END_GET
END_PROPERTY

PROPERTY P_sBufferType : STRING
SET
sBufferType := P_sBufferType;
END_SET
END_PROPERTY

END_FUNCTION_BLOCK

// ---- ECC/Tools/LogToFile/FB_LogToFile.TcPOU
FUNCTION_BLOCK FB_LogToFile
VAR_INPUT
END_VAR
VAR_OUTPUT
	Busy : BOOL;
END_VAR
VAR
	State:INT;
	StateDelFile:INT;
	StateSetDate:INT;
	msg_old : STRING(200);
	msgWithTime : STRING(255);
	msgToWrite : STRING(3000);
	tmpMsgToWrite : STRING(3000);
	StateOld:INT;
	hFileOld:UINT;

	OpenFile:FB_FileOpen;
	WriteFile:FB_FileWrite;
	CloseFile:FB_FileClose;
	DeleteFile:FB_FileDelete;
	CurrentDate:STRING(10);
	PathAndFile:STRING(200);

	PathAndFileDelete:STRING(200);

	(*Control and status *)

	bFileOpenError:BOOL;
	nFileOpenErrorID:UDINT;
	hFile:UINT;

	bFileWriteError:BOOL;
	nFileWriteErrorID:UDINT;

	bFileCloseError:BOOL;
	nFileCloseErrorID:UDINT;
	nFileCloseError: BOOL;

	nDeleteFileErrorID:UDINT;
	bDeleteFileError:BOOL;

	DateTimeNow		:STRING;
	DateNow			:STRING(10);

	CPUCOUNTER: GETCPUCOUNTER;
	Scan_EndMeassurement:DWORD;
	Scan_EndMeassurementHigh:DWORD;
	Scan_Current_us:DWORD;
	CPUScanLimitReach:BOOL;

	CPUScanLimOld:BOOL;

	MaxEntriesFifo:INT;
	SetFifoLog:FB_SetFifo;
	GetFifoLog:FB_GetFifo;

	i:INT;
	Sourcepointer: POINTER TO STRING(3000);//DWORD;
	DestPointer:POINTER TO STRING(3000);//DWORD;
	SourceLength:INT;
	DestLength:DWORD;
	TotalLength:INT;
	MaxTotalLength:INT;

	DateChanged:BOOL;
	DelYear:INT;
	DelMonth:INT;
	DelDay:INT;
	DelMonthString:STRING(2);
	TempString:STRING;
	OS_Error:BOOL;

	(* Use as setting for example from XML settings *)
	EnableHouseKeeping:BOOL:=TRUE;	(* Enable/disable housekeeping *)
	LogStoreDays:INT:=7;			(* How many days to keep logs *)
	NumberOfTries:INT:=7;			(* How many days before to try to delete. To double check cleaning *)
	ErrorCount:INT;
END_VAR
VAR PERSISTENT 
// Log to file
	DaysOfLog 			: INT:=14;
END_VAR

(* Monitor system resources and stop write to log if scantime exceeded *)
//A_SystemMonitor();

//File logging
fbLocalTime(
	sNetID:= '', 
	bEnable:= TRUE, 
	dwCycle:= 5, 
	dwOpt:= 0, 
	tTimeout:=DEFAULT_ADS_TIMEOUT );	

(* Check buffer for text stream to write to file *)
A_WriteToLog();

(* Execute housekeeping if date changed *)
A_Housekeeping();

ACTION A_Housekeeping:
(* Change number of days to log *)
IF (DaysOfLog > 0) THEN
	LogStoreDays := DaysOfLog;
END_IF

(* Housekeeping: Delete files from x numbers of days back *)
IF DateChanged AND StateSetDate = 0 AND EnableHouseKeeping THEN
	DelYear := STRING_TO_INT(MID(CurrentDate, 4, 1));
	DelMonth := STRING_TO_INT(MID(CurrentDate, 2, 6));
	DelDay := STRING_TO_INT(MID(CurrentDate, 2, 9));

	(* Set start date and wrap around month + year if needed *)
	IF DelDay <= LogStoreDays THEN
		DelDay := 31 + DelDay - LogStoreDays;
		DelMonth := DelMonth - 1;
	ELSE
		DelDay := DelDay - LogStoreDays;
	END_IF

	IF DelMonth < 1 THEN
		DelMonth := DelMonth + 12;
		DelYear := DelYear - 1;
	END_IF

	StateSetDate := 1;

ELSIF DateChanged AND StateDelFile = 9999 THEN
	F_LogFile('WARNING: Housekeep stopped');
	DateChanged := FALSE;
ELSIF NOT EnableHouseKeeping THEN
	DateChanged := FALSE;
END_IF

CASE StateSetDate OF
	0: (* Do nothing *)
		;
	1: (* Initialize *)
		DateChanged := FALSE;
		StateSetDate := StateSetDate + 1;
		ErrorCount := 0;

		F_LogFile('LogToFile - Housekeep - New day!!');
		F_LogFile(Tempstring);

	2: (* Set Date to delete *)

		(* Combine to file and path *)
		PathAndFileDelete := CONCAT('C:\Log\', INT_TO_STRING(DelYear));
		PathAndFileDelete := CONCAT(PathAndFileDelete, '-');
		PathAndFileDelete := CONCAT(PathAndFileDelete, F_PadWith(DelMonth, 2, '0'));
		PathAndFileDelete := CONCAT(PathAndFileDelete, '-');
		PathAndFileDelete := CONCAT(PathAndFileDelete, F_PadWith(DelDay, 2, '0'));
		PathAndFileDelete := CONCAT(PathAndFileDelete, ' PLC Debug.txt');


		OS_Error := FALSE;
		StateDelFile := 1;
		StateSetDate := StateSetDate + 1;

		TempString := 'LogToFile - Housekeep: ';
		TempString := CONCAT('Try to delete: ', PathAndFileDelete);
		TempString := CONCAT(TempString, ' And ');
		TempString := CONCAT(TempString, INT_TO_STRING(NumberOfTries - ErrorCount));
		TempString := CONCAT(TempString, ' days before');
		F_LogFile(Tempstring);


	3: (* Wait for file deletion to complete *)
		IF ErrorCount < NumberOfTries AND StateDelFile = 0 THEN

			(* Set start date and wrap around month + year if needed *)
			IF DelDay - 1 <= 0 THEN
				DelDay := 31;
				DelMonth := DelMonth - 1;
			ELSE
				DelDay := DelDay - 1;
			END_IF

			IF DelMonth < 1 THEN
				DelMonth := DelMonth + 12;
				DelYear := DelYear - 1;
			END_IF

			StateSetDate := 2;

		ELSIF ErrorCount >= NumberOfTries AND StateDelFile = 0 THEN
			StateSetDate := 0;

			F_LogFile('LogToFile - Housekeep: Done deleting file(s)');
		END_IF

END_CASE

CASE StateDelFile OF

	0: (* Do nothing*)
		;
	1: (* Delete root file *)

		DeleteFile( bExecute := FALSE );

		DeleteFile(
		sNetId:= '',
		sPathName:= PathAndFileDelete,
		ePath:= PATH_GENERIC,
		bExecute:= TRUE,
		tTimeout:= t#3s,
		);

		StateDelFile := StateDelFile + 1;


	2: (* Wait for not busy and check for error *)
		DeleteFile( bExecute := FALSE );

		IF NOT DeleteFile.bBusy THEN
			IF DeleteFile.bError THEN
				nDeleteFileErrorID := DeleteFile.nErrId;
				bDeleteFileError := TRUE;
				StateDelFile := 9999;

			ELSE
				StateDelFile:= 0;
				ErrorCount := 0;

				TempString := ('LogToFile - Housekeep: Deleted file: ');
				TempString := CONCAT(TempString, PathAndFileDelete);
				F_LogFile(TempString);
			END_IF
		END_IF

	9999: (* FileDelete error *)
		IF nDeleteFileErrorID = 1804 THEN (* File not found *)
			F_LogFile('LogToFile - Housekeep: File not found - ignore');
			nDeleteFileErrorID := 0;
			bDeleteFileError := FALSE;
			StateDelFile:= 0;
			ErrorCount := ErrorCount + 1;
		ELSE (* Any other error *)

			IF NOT OS_Error THEN
				TempString := ('LogToFile - Housekeep: Failed with ADS errorID: ');
				TempString := CONCAT(TempString, UDINT_TO_STRING(nDeleteFileErrorID));
				F_LogFile(TempString);
				OS_Error := TRUE;
			END_IF
		END_IF
	END_CASE
END_ACTION

ACTION A_SystemMonitor:
(* Check for new log stream and put into FIFO buffer with time stamp *)

(* Calculate current time of scan *)
	CPUCOUNTER(cpuCntLoDW=>Scan_EndMeassurement , cpuCntHiDW=>Scan_EndMeassurementHigh );
	Scan_Current_us:=(Scan_EndMeassurement-MAIN.TimeStamps.StartMeassurement)/10000;

	(* Did we have a warning ?*)
	IF Scan_Current_us > Util.Scan_Warning_us THEN
		CPUScanLimitReach := TRUE;

		IF NOT CPUScanLimOld THEN
			(* Get date and time *)
			DateTimeNow  := TO_STRING(SYSTEMTIME_TO_DT(timestr:=MAIN.fbLocalTime.systemTime));

			(* Set date to check for generation of new file *)
			CurrentDate := DateTimeNow;

			(* Add date and time to line of log *)
			msgWithTime := CONCAT(DateTimeNow, ' ');
			msgWithTime := CONCAT(msgWithTime, 'Maximum scan time exceeded - File logging to disk paused!!');
			msgWithTime := CONCAT(msgWithTime, '$N');

			SetFifoLog(
				in_STRING:= msgWithTime,
				in_Owner:= 'LogToFile',
				in_LogLevel:= 0,
				DB:= LogToTextBuffer);

			CPUScanLimOld := TRUE;
		END_IF
	ELSE
		IF CPUScanLimOld THEN
			(* Get date and time *)
			DateTimeNow  := Get_SystemTime();

			CurrentDate := DateTimeNow;

			(* Add date and time to line of log *)
			msgWithTime := CONCAT(DateTimeNow, ' ');
			msgWithTime := CONCAT(msgWithTime, 'File logging resumed');
			msgWithTime := CONCAT(msgWithTime, '$N');

			SetFifoLog(
				in_STRING:= msgWithTime,
				in_Owner:= 'LogToFile',
				in_LogLevel:= 0,
				DB:= LogToTextBuffer);
		END_IF

		CPUScanLimitReach := FALSE;
		CPUScanLimOld := FALSE;
	END_IF

IF LogToTextBuffer.Count > MaxEntriesFifo THEN
	MaxEntriesFifo := LogToTextBuffer.Count;
END_IF
END_ACTION

ACTION A_WriteToLog:
(* Ready for new logline to be written *)
IF State = 0 AND LogToTextBuffer.Count > 0 AND NOT CPUScanLimitReach THEN

	(* Get date and time *)
	DateTimeNow  := SYSTEMTIME_TO_STRING(fbLocalTime.systemTime);

	(* New date - set flag for housekeeping *)
	DateNow := DateTimeNow;
	IF CurrentDate <> DateNow THEN
		DateChanged := TRUE;
	END_IF

	(* Set date to check for generation of new file *)
	CurrentDate := DateTimeNow;

	(* Set Path and filename *)
	PathAndFile := 'C:\Log\';
	PathAndFile := CONCAT(PathAndFile, CurrentDate);
	PathAndFile := CONCAT(PathAndFile, ' PLC Debug');
	PathAndFile := CONCAT(PathAndFile, '.txt');

	State := 1;
	Busy := TRUE;
END_IF

CASE State OF

0:	(* Do nothing *)
	;

1: (* Open File *)

	OpenFile( bExecute := FALSE );

	OpenFile(
		sNetId:= '',
		sPathName:= PathAndFile,
		nMode:= FOPEN_MODEAPPEND,
		ePath:= PATH_GENERIC,
		bExecute:= TRUE,
		tTimeout:= t#3s,
		);

	State := State +1;

2: (* Wait for not busy - check for error *)

	OpenFile( bExecute := FALSE );

	IF NOT OpenFile.bBusy THEN

		IF OpenFile.bError THEN
			nFileOpenErrorID := OpenFile.nErrId;
			bFileOpenError := TRUE;
			State := 50;
		ELSE
			hFile := OpenFile.hFile;
			State := State + 1;
		END_IF
	END_IF


3: (* Put line into file *)

	WriteFile ( bExecute := FALSE );

	msgToWrite := '';
	DestLength := 0;
	TotalLength := 0;
	SourcePointer := ADR(tmpMsgToWrite);
	DestPointer := ADR(msgToWrite);

	(* Bundle to maximum 2700 + logline amount of bytes *)
	WHILE TotalLength < 2700 AND LogToTextBuffer.Count > 0 DO

		GetFifoLog(
			DB:= LogToTextBuffer,
			out_STRING=> );

		tmpMsgToWrite := GetFifoLog.out_STRING;
		SourceLength := LEN(tmpMsgToWrite);
		TotalLength := SourceLength + TotalLength;
  		MEMCPY (DestPointer, SourcePointer, SourceLength);

		Destpointer := DestPointer + SourceLength;

	END_WHILE

	(* Save maximum totallengt of string to write to file for debug use *)
	IF TotalLength > MaxTotalLength THEN
		MaxTotalLength := TotalLength;
	END_IF

	WriteFile(
	sNetId:= '',
	hFile:= hFile,
	pWriteBuff:= ADR(msgToWrite),
	cbWriteLen:= TotalLength,
	bExecute:= TRUE,
	tTimeout:= t#3s,
	);

	State := State + 1;

4: (* Wait for not busy and check for error *)

	WriteFile( bExecute := FALSE );

	IF NOT WriteFile.bBusy THEN
		IF WriteFile.bError THEN
			nFileWriteErrorID := WriteFile.nErrId;
			bFileWriteError := TRUE;
			State := 50;
		ELSE
			State := State + 1;
		END_IF
	END_IF


5: (* Close file *)

	CloseFile( bExecute := FALSE );

	CloseFile(
		sNetId:= '',
		hFile:= hFile,
		bExecute:= TRUE,
		tTimeout:= t#3s,
		);

	State := State + 1;

6: (* Wait for not busy and check for error *)

	CloseFile( bExecute := FALSE );

	IF NOT CloseFile.bBusy THEN
		IF CloseFile.bError THEN
			nFileCloseErrorID := CloseFile.nErrId;
			bFileCloseError := TRUE;
		END_IF

		State := 50;
		hFile := 0;
	END_IF

50: (* Error or ready => Cleanup *)

	IF hFile <> 0 THEN
		State := 5; (* Close the file *)
	ELSE
		State := 0;
		Busy := FALSE;
	END_IF

END_CASE
END_ACTION

END_FUNCTION_BLOCK

// ---- ECC/Tools/LogToFile/FB_SetFifo.TcPOU
FUNCTION_BLOCK FB_SetFifo
VAR_INPUT
	in_STRING:STRING(255);
END_VAR
VAR_OUTPUT
	bFIFO_Full:BOOL;
END_VAR
VAR_IN_OUT
	DB:ST_String_FIFO;
END_VAR
VAR
	TempString:STRING(255);
END_VAR

(* Insert data to fifo*)
bFIFO_Full := FALSE;
IF DB.Count <= DB.DataTop THEN

	(* Calculate new insert pointer *)
	DB.Input_Pointer := DB.Input_Pointer + 1;
	IF DB.Input_Pointer > DB.DataTop THEN
		DB.Input_Pointer := 0;
	END_IF

	(* If data is impty, sync output pointer *)
	IF DB.Count = 0 THEN
		DB.Output_Pointer := DB.Input_Pointer;
	END_IF

	(* Store data *)
	DB.DB[DB.Input_Pointer] := in_STRING;

	DB.Count := DB.Count + 1;

ELSE
	bFIFO_Full := TRUE;
END_IF

END_FUNCTION_BLOCK

// ---- ECC/Tools/LogToFile/FB_GetFifo.TcPOU
FUNCTION_BLOCK FB_GetFifo
VAR_INPUT
END_VAR
VAR_OUTPUT
	bFIFO_Empty:BOOL;
	out_STRING:STRING(255);
END_VAR
VAR_IN_OUT
	DB:ST_String_FIFO;
END_VAR
VAR
END_VAR

bFIFO_Empty := FALSE;
IF DB.Count > 0 THEN
	out_STRING := DB.DB[DB.Output_Pointer];
	DB.DB[DB.Output_Pointer] := '';
	DB.Count := DB.Count - 1;

	DB.Output_Pointer := DB.Output_Pointer + 1;
	IF DB.Output_Pointer > DB.DataTop THEN
		DB.Output_Pointer := 0;
	END_IF

ELSE
	bFIFO_Empty := TRUE;
END_IF

END_FUNCTION_BLOCK

// ---- ECC/Tools/LogToFile/F_PadWith.TcPOU
FUNCTION F_PadWith : STRING
VAR_INPUT
	in_Int:INT;
	in_NumOfBytes:INT;
	in_PadWith:STRING;
END_VAR
VAR
	i:INT;
	TempString:STRING;
END_VAR

TempString := '';

FOR i := 1 TO in_NumOfBytes - LEN(INT_TO_STRING(in_INT)) DO
	TempString := CONCAT(TempString, in_PadWith);
END_FOR

F_PadWith := CONCAT(TempString, INT_TO_STRING(in_INT));

END_FUNCTION

// ---- ReadConfigFile/FB_ReadFile.TcPOU
FUNCTION_BLOCK FB_ReadFile

VAR
	CSVMemBufferReader		:FB_CSVMemBufferReader;
	fbFileOpen				:FB_FileOpen;
	fbFileGet				:FB_FileGets;
	fbFileClose				:FB_FileClose;
	
//	sPathName				:STRING := 'C:\RUO folder\Configuration file branches TEST\';
//	sFileName				:STRING := 'NEW TEST\test-branches-config-file\config';
//	sConfigPathFile			:STRING(300) := CONCAT(sPathName, sFileName);
	sConfigPathFile			:STRING(300) := 'C:\config\config';
	
	bReset					:BOOL;
	nCol					:INT;
	hFile					:UINT;
	value					:STRING[300];
	sBufferString			:ARRAY[0..15]OF STRING;
	iStep					:INT;
	sLine					:STRING;
	nRow					:INT;
	bRead					:BOOL := TRUE;
	bEOF					:BOOL;
	i						:INT;
	iCRLFCounter			:INT;
	
	// split string
	aSplit					:ARRAY[0..cMax] OF STRING(255);
	bResultSplit			:BOOL;
	ii						:UDINT;
END_VAR
VAR CONSTANT
	cStepInit				:INT := 0;
	cStepOpenFile			:INT := 10;
	cStepGetLine			:INT := 20;
	cStepEOFCheck			:INT := 25;
	cStepReadLine			:INT := 30;
	cStepParseData			:INT := 35;
	cStepCloseFile			:INT := 40;
	cStepError				:INT := 8000;
	
	// split string
	cMax					:UDINT := 15;
END_VAR

(*
	TEST OF ONLINE CHANGES WITH MERGE BRANCHES
*)
(*
	TEST OF ONLINE CHANGES WITH MERGE BRANCHES
*)
(*
	TEST OF ONLINE CHANGES WITH MERGE BRANCHES
*)

CASE iStep OF
	
	cStepInit:
	
		//* semicolon (;) := 16#3B => german field separator, comma (,) := 16#2C => US field separator
		DEFAULT_CSV_FIELD_SEP := 16#3B;
		
		nRow := 0;
		nCol := 0;
		iCRLFCounter := 0;
		bEOF := FALSE;
		bReset := FALSE;
		
		// fb Reset
		fbFileOpen(bExecute := FALSE);
		fbFileClose(bExecute := FALSE);
		fbFileGet(bExecute := FALSE);
			
		IF bRead 
			AND NOT fbfileopen.bBusy
			AND NOT fbfileclose.bBusy
			AND NOT fbfileget.bBusy
			THEN
			
			FOR i := 0 TO 24 DO
				GVL.sString[i] := '';
				
			END_FOR
			iStep := cStepOpenFile;
			bRead := FALSE;
		END_IF;
		
		cStepOpenFile:
			fbFileopen(	sNetId := '', sPathName := sConfigPathFile, nMode := FOPEN_MODEREAD,
						ttimeout := T#3S, ePath := E_OpenPath.PATH_GENERIC, bExecute := TRUE, hFile => hfile);
					
		IF NOT fbfileopen.bBusy THEN
			IF fbfileopen.bError THEN
				iStep := cStepError;	
			ELSE
				iStep := cStepGetLine;
			END_IF
		END_IF
		
		cStepGetLine:
			fbFileGet(hFile := hFile, bExecute := TRUE, sLine => sLine);
	
		IF NOT fbFileGet.bBusy THEN
			IF fbFileGet.bError THEN
				iStep := cStepError;	
			ELSE IF fbFileGet.bEOF THEN
				bEOF := TRUE;
			END_IF
		(*
			IF RIGHT( Fileget.sLine, 1 ) = '$N' THEN
				sCSVLine := REPLACE( sCSVLine, '$R$L', 2, LEN( sCSVLine ) );
			END_IF
		*)
			iStep := cStepEOFCheck;
			END_IF
		END_IF
		
		cStepEOFCheck:
				fbFileGet(bExecute := FALSE);
		IF bEOF THEN
			iStep := cStepCloseFile;
		ELSE
			iStep := cStepReadLine;	
		END_IF
	
		cStepReadLine:
			nCol := 0;
			CSVMemBufferReader.eCmd := E_EnumCmdType.eEnumCmd_First;
				REPEAT
					CSVMemBufferReader(pBuffer := ADR(sLine), cbBuffer := SIZEOF(sLine), getValue => value);
				
					IF CSVMemBufferReader.bOk THEN
						sBufferString[ncol] := value;
						CSVMemBufferReader.eCmd := E_EnumCmdType.eEnumCmd_Next;
						ncol := ncol + 1;
						IF CSVMemBufferReader.bCRLF THEN
							iCRLFCounter := iCRLFCounter + 1;
						END_IF
					END_IF
				UNTIL NOT CSVMemBufferReader.bOk 
				END_REPEAT	
			istep := cStepParseData;
			
		cStepParseData:
			// check EOF
			IF fbFileGet.bEOF THEN
				iStep := cStepCloseFile;
			ELSE
				GVL.sString[nRow] := sBufferString[0];
				nRow := nRow + 1;
				iStep := cStepGetLine;
			END_IF
		
		cStepCloseFile:	
			fbFileClose(hFile := hFile, bExecute := TRUE);
			IF NOT fbFileClose.bBusy THEN
				IF fbFileClose.bError THEN
					iStep := cStepError;	
				END_IF
			ELSE
				fbFileClose(bExecute:=FALSE);
				iStep := cStepInit;
			END_IF
			
		cStepError:
			IF bReset THEN
				iStep := cStepInit;
			END_IF
END_CASE

// split/parse strings
FOR ii := 0 TO cMax - 1 DO
	
	aSplit[ii] := GVL.sString[ii];
	bResultSplit := FindAndSplitChar(sSeparatorChar := '=', pSrcString := ADR(aSplit[ii]),
									  pLeftString := ADR(aSplit[ii + 1]), nLeftSize := SIZEOF(aSplit[ii + 1]),
									  pRightString := ADR(aSplit[ii]), nRightSize := SIZEOF(aSplit[ii]),
									  bSearchFromRight := FALSE);
									  
	// assign values from config file
	GVL.sVars.sEnvironment		:= aSplit[0];
	GVL.sVars.sCellName			:= aSplit[1];
	GVL.sVars.sIpAddress 		:= aSplit[2];
	GVL.sVars.sAmsNetId 		:= aSplit[3];
	GVL.sVars.sOpcUaURL 		:= aSplit[4];
	GVL.sVars.sStation1			:= aSplit[5];
	GVL.sVars.sTrackserver		:= aSplit[6];
	GVL.sVars.sTrackserver_AMS	:= aSplit[7];
	
//	GVL.sVars.sUhfRfidOpcUaURL 	:= aSplit[5];
//	GVL.sVars.sHfRfidOpcUaURL 	:= aSplit[6];
//	GVL.sVars.sStation2			:= aSplit[8];
//	GVL.sVars.sStation3			:= aSplit[9];
//	GVL.sVars.sStation4			:= aSplit[10];
//	GVL.sVars.sRelease			:= aSplit[11];
//	GVL.sVars.sTag				:= aSplit[12];
	
	IF NOT bResultSplit THEN
		EXIT;
	END_IF
END_FOR

END_FUNCTION_BLOCK

// ---- ECC/Basic/Common Units/FB_Units.TcPOU
// Common unit codes and symbols are taken from document:
// rec20_Rev13e_2017.xls 
FUNCTION_BLOCK FB_Units
VAR_INPUT
END_VAR
VAR_OUTPUT
END_VAR
VAR CONSTANT
	MAXSIZE		: BYTE := 50;
END_VAR
VAR
	// array of possible unitcodes/units
	aUnits		: ARRAY [0..MAXSIZE, 0..1] OF STRING(10);
	bInitDone	: BOOL;
END_VAR


M_Init();

METHOD PUBLIC Code : STRING
VAR_INPUT
	eUnit		: E_Units;
END_VAR
/// Returns the common unit code for the definded unit type

// Make sure valuesa are initialized
M_Init();

IF (eUnit <= MAXSIZE) THEN
	Code := aUnits[eUnit, 0];	

ELSE
	Code := aUnits[0, 0];

END_IF
END_METHOD

METHOD PROTECTED M_Init
VAR_INPUT
END_VAR
VAR
	i		: BYTE;
END_VAR
// Add the units needed
// NOTE: Must match the enumeration E_CommonUnits!!
IF (NOT bInitDone) THEN
	i := 0;
	// Init with selectable units
	aUnits[i, 0] := '';		aUnits[i, 1] := '';			i := i+1;	// Empty / fallback

	aUnits[i, 0] := 'MTR';	aUnits[i, 1] := 'm';		i := i+1;
	aUnits[i, 0] := 'CMT';	aUnits[i, 1] := 'cm';		i := i+1;
	aUnits[i, 0] := 'MMT';	aUnits[i, 1] := 'mm';		i := i+1;
	aUnits[i, 0] := '4H';	aUnits[i, 1] := 'µm';		i := i+1;
	aUnits[i, 0] := 'C45';	aUnits[i, 1] := 'nm';		i := i+1;

	aUnits[i, 0] := 'KGM';	aUnits[i, 1] := 'kg';		i := i+1;
	aUnits[i, 0] := 'GRM';	aUnits[i, 1] := 'g';		i := i+1;

	aUnits[i, 0] := 'M46';	aUnits[i, 1] := 'r/min';	i := i+1;
	aUnits[i, 0] := 'C16';	aUnits[i, 1] := 'mm/s';		i := i+1;
	aUnits[i, 0] := 'H81';	aUnits[i, 1] := 'mm/min';	i := i+1;
	aUnits[i, 0] := 'MTS';	aUnits[i, 1] := 'm/s';		i := i+1;
	aUnits[i, 0] := '2X';	aUnits[i, 1] := 'm/min';	i := i+1;
	
	aUnits[i, 0] := 'M41';	aUnits[i, 1] := 'mm/s²';	i := i+1;

	aUnits[i, 0] := 'P1';	aUnits[i, 1] := '%';		i := i+1;	
	
	aUnits[i, 0] := 'DD';	aUnits[i, 1] := '°';		i := i+1;	
	aUnits[i, 0] := 'CEL';	aUnits[i, 1] := '°C';		i := i+1;	
	aUnits[i, 0] := 'FAH';	aUnits[i, 1] := '°F';		i := i+1;	

	aUnits[i, 0] := 'BAR';	aUnits[i, 1] := 'bar';		i := i+1;	

	aUnits[i, 0] := 'DAY';	aUnits[i, 1] := 'day';		i := i+1;	
	aUnits[i, 0] := 'HUR';	aUnits[i, 1] := 'h';		i := i+1;	
	aUnits[i, 0] := 'MIN';	aUnits[i, 1] := 'min';		i := i+1;	
	aUnits[i, 0] := 'SEC';	aUnits[i, 1] := 's';		i := i+1;	
	aUnits[i, 0] := 'C26';	aUnits[i, 1] := 'ms';		i := i+1;	
	aUnits[i, 0] := 'B98';	aUnits[i, 1] := 'µs';		i := i+1;	
	aUnits[i, 0] := 'C47';	aUnits[i, 1] := 'ns';		i := i+1;	

	aUnits[i, 0] := '2G';	aUnits[i, 1] := 'V';		i := i+1;	
	aUnits[i, 0] := '2H';	aUnits[i, 1] := 'V';		i := i+1;	
	aUnits[i, 0] := '2Z';	aUnits[i, 1] := 'mV';		i := i+1;	
	aUnits[i, 0] := 'AMP';	aUnits[i, 1] := 'A';		i := i+1;	
	aUnits[i, 0] := '4K';	aUnits[i, 1] := 'mA';		i := i+1;	
	aUnits[i, 0] := 'B84';	aUnits[i, 1] := 'µA';		i := i+1;	
	aUnits[i, 0] := 'KWH';	aUnits[i, 1] := 'KWh';		i := i+1;	
	aUnits[i, 0] := 'KWT';	aUnits[i, 1] := 'KW';		i := i+1;	
	aUnits[i, 0] := 'WTT';	aUnits[i, 1] := 'W';		i := i+1;	
	aUnits[i, 0] := 'C31';	aUnits[i, 1] := 'mW';		i := i+1;	
	aUnits[i, 0] := 'D80';	aUnits[i, 1] := 'µW';		i := i+1;	

	aUnits[i, 0] := 'MHZ';	aUnits[i, 1] := 'MHz';		i := i+1;	
	aUnits[i, 0] := 'KHZ';	aUnits[i, 1] := 'kHz';		i := i+1;	
	aUnits[i, 0] := 'HTZ';	aUnits[i, 1] := 'Hz';		i := i+1;	

	bInitDone := TRUE;
	
END_IF
END_METHOD

METHOD PUBLIC Text : STRING
VAR_INPUT
	eUnit		: E_Units;
END_VAR
/// Returns the common unit code for the definded unit type

// Make sure valuesa are initialized
M_Init();

IF (eUnit <= MAXSIZE) THEN
	Text := aUnits[eUnit, 1];	

ELSE
	Text := aUnits[0, 1];

END_IF
END_METHOD

END_FUNCTION_BLOCK

// ---- ECC/Components/FB_AI.TcPOU
FUNCTION_BLOCK FB_AI EXTENDS FB_Basic
VAR_OUTPUT
	rValue		: LREAL;
END_VAR
VAR
	fbLinTrafo	: FB_LIN_TRAFO;

// HW
	Status AT %I* : WORD;		// Status word from IO module
	{attribute 'OPC.UA.DA':='1'}
	{attribute 'OPC.UA.DA.Access' := '1'}
	{attribute 'OPC.UA.DA.Description' := 'Input I/O signal (RAW)'}
	{attribute 'OPC.UA.DA.StructuredType' := '0'}
	Value AT %I* : INT;			// Value from IO module
	State AT %I* : WORD := 8;	// State from Ethercat module
	AdsAdrr AT %I* : AMSADDR;	// ADS address from EtherCAT module

END_VAR
VAR PERSISTENT
	rScaleMax	: LREAL := 100;
	rScaleMin	: LREAL := -100;
	bUseLoLo	: BOOL;
	rLoLo		: LREAL := -100;
	bUseLo		: BOOL;
	rLo			: LREAL := -100;
	bUseHi		: BOOL;
	rHi			: LREAL := 100;
	bUseHiHi	: BOOL;
	rHiHi		: LREAL := 100;

END_VAR


// Run parent FB
SUPER^();

METHOD PROTECTED M_AutoMode : BOOL
VAR_INPUT
END_VAR
// Analog inputs automatic mode
// Executed from parent FB_Basic

IF (P_bEnable) THEN
	rActualValue := rAutoValue;
ELSE
	rActualValue := 0.0;
END_IF

rValue := rActualValue;
END_METHOD

METHOD PROTECTED M_ErrorHandling : BOOL
VAR_INPUT
END_VAR
// Error handling
IF (bCmdEnable) THEN
	IF (NOT P_bManualMode) THEN
		// Hardware errors
		IF (NOT F_ECat_OK(State)) THEN
			// EtherCAT state
			bStaError := TRUE;
			eStaErrorID := E_ComponentErrors.HW_ECat_Not_OP;
		ELSIF (Status.14) THEN
			// Module internal error
			bStaError := TRUE;
			eStaErrorID := E_ComponentErrors.HW_Internal_Error;
		ELSIF (Status.0) THEN
			// Underrange
			bStaError := TRUE;
			eStaErrorID := E_ComponentErrors.HW_UnderRange;
		ELSIF (Status.1) THEN
			// Overrange
			bStaError := TRUE;
			eStaErrorID := E_ComponentErrors.HW_OverRange;
		ELSIF (Status.2) THEN
			// Limit1
			bStaError := TRUE;
			eStaErrorID := E_ComponentErrors.HW_Limit1;
		ELSIF (Status.2) THEN
			// Limit2
			bStaError := TRUE;
			eStaErrorID := E_ComponentErrors.HW_Limit2;
		END_IF
	END_IF
	
	// Software errors
	IF (bUseHiHi AND (rActualValue > rHiHi)) THEN
		bStaError := TRUE;
		eStaErrorID := E_ComponentErrors.SW_HiHi;
	END_IF
	IF (bUseHi AND (rActualValue > rHi)) THEN
		bStaWarning := TRUE;
		eStaErrorID := E_ComponentErrors.SW_Hi;
	END_IF
	IF (bUseLoLo AND (rActualValue < rLolo)) THEN
		bStaError := TRUE;
		eStaErrorID := E_ComponentErrors.SW_LoLo;
	END_IF
	IF (bUseLo AND (rActualValue < rLo)) THEN
		bStaWarning := TRUE;
		eStaErrorID := E_ComponentErrors.SW_Lo;
	END_IF
	
ELSE
	bStaError := FALSE;
	bStaWarning := FALSE;
	eStaErrorID := E_ComponentErrors.OK;

END_IF
END_METHOD

METHOD PROTECTED M_Init : BOOL
VAR_INPUT
END_VAR
// Init

bCmdEnable := TRUE;
bInitDone := TRUE;
END_METHOD

METHOD PROTECTED M_ManualMode : BOOL
VAR_INPUT
END_VAR
// Analog inputs manual mode
// Executed from parent FB_Basic

rManualValue := LIMIT(rScaleMin, rManualValue, rScaleMax);

IF (P_bEnable) THEN
	rActualValue := rManualValue;
ELSE
	rActualValue := 0.0;
END_IF

rValue := rActualValue;
END_METHOD

METHOD PROTECTED M_Run : BOOL
VAR_INPUT
END_VAR
// Analog inputs run
// Executed from parent FB_Basic

// Update IO 

fbLinTrafo(	rIN := Value,
			rIN_MIN := -32767,
			rIN_MAX := 32767,
			rOUT_MIN := rScaleMin,
			rOUT_MAX := rScaleMax,
			rOUT => rAutoValue,
			bERROR =>	);
END_METHOD

END_FUNCTION_BLOCK

// ---- ECC/Components/FB_Basic.TcPOU
FUNCTION_BLOCK FB_Basic
VAR_INPUT
END_VAR
VAR_OUTPUT
END_VAR
VAR
// Commands
	{attribute 'OPC.UA.DA':='1'}
	{attribute 'OPC.UA.DA.Access' := '3'}
	{attribute 'OPC.UA.DA.Description' := 'Enable component'}
	{attribute 'OPC.UA.DA.StructuredType' := '0'}
	bCmdEnable		: BOOL;		// Write from e.g. HMI
	{attribute 'OPC.UA.DA':='1'}
	{attribute 'OPC.UA.DA.Access' := '3'}
	{attribute 'OPC.UA.DA.Description' := 'Enable manual mode'}
	{attribute 'OPC.UA.DA.StructuredType' := '0'}
	bCmdManual		: BOOL;		// Write from e.g. HMI
	{attribute 'OPC.UA.DA':='1'}
	{attribute 'OPC.UA.DA.Access' := '3'}
	{attribute 'OPC.UA.DA.Description' := 'Enable automatic mode'}
	{attribute 'OPC.UA.DA.StructuredType' := '0'}
	bCmdAuto		: BOOL;		// Write from e.g. HMI
	{attribute 'OPC.UA.DA':='1'}
	{attribute 'OPC.UA.DA.Access' := '3'}
	{attribute 'OPC.UA.DA.Description' := 'Reset component'}
	{attribute 'OPC.UA.DA.StructuredType' := '0'}
	bCmdReset		: BOOL;		// Write from PLC or HMI to reset errors and warnings
	
// Status
	{attribute 'OPC.UA.DA':='1'}
	{attribute 'OPC.UA.DA.Access' := '1'}
	{attribute 'OPC.UA.DA.Description' := 'Running status'}
	{attribute 'OPC.UA.DA.StructuredType' := '0'}
	bStaRunning		: BOOL;
	{attribute 'OPC.UA.DA':='1'}
	{attribute 'OPC.UA.DA.Access' := '1'}
	{attribute 'OPC.UA.DA.Description' := 'Error status'}
	{attribute 'OPC.UA.DA.StructuredType' := '0'}
	bStaError		: BOOL;
	{attribute 'OPC.UA.DA':='1'}
	{attribute 'OPC.UA.DA.Access' := '1'}
	{attribute 'OPC.UA.DA.Description' := 'Error ID'}
	{attribute 'OPC.UA.DA.StructuredType' := '0'}
	eStaErrorID		: E_ComponentErrors;
	{attribute 'OPC.UA.DA':='1'}
	{attribute 'OPC.UA.DA.Access' := '1'}
	{attribute 'OPC.UA.DA.Description' := 'Warning status'}
	{attribute 'OPC.UA.DA.StructuredType' := '0'}
	bStaWarning		: BOOL;
	{attribute 'OPC.UA.DA':='1'}
	{attribute 'OPC.UA.DA.Access' := '1'}
	{attribute 'OPC.UA.DA.Description' := 'Manual mode enabled'}
	{attribute 'OPC.UA.DA.StructuredType' := '0'}
	bStaManual		: BOOL;
	bInitDone		: BOOL;

// Values
	{attribute 'OPC.UA.DA':='1'}
	{attribute 'OPC.UA.DA.Access' := '3'}
	{attribute 'OPC.UA.DA.Description' := 'Manual value'}
	{attribute 'OPC.UA.DA.StructuredType' := '0'}
	rManualValue	: LREAL;	// Write from e.g. HMI
	rAutoValue		: LREAL;	// Write from program
	{attribute 'OPC.UA.DA':='1'}
	{attribute 'OPC.UA.DA.Access' := '1'}
	{attribute 'OPC.UA.DA.Description' := 'Actual value'}
	{attribute 'OPC.UA.DA.StructuredType' := '0'}
	rActualValue	: LREAL;
	
	trigManOn		: R_TRIG;
	trigAutoOn		: R_TRIG;

END_VAR
VAR PERSISTENT
	{attribute 'OPC.UA.DA':='1'}
	{attribute 'OPC.UA.DA.Access' := '1'}
	{attribute 'OPC.UA.DA.Description' := 'Component tag'}
	{attribute 'OPC.UA.DA.StructuredType' := '0'}
	sTag			: STRING;
	{attribute 'OPC.UA.DA':='1'}
	{attribute 'OPC.UA.DA.Access' := '1'}
	{attribute 'OPC.UA.DA.Description' := 'Component name'}
	{attribute 'OPC.UA.DA.StructuredType' := '0'}
	sName			: STRING;
END_VAR


// Run methods (overwrite in inherited FB's)
IF (NOT bInitDone) THEN
	M_Init();
ELSE
	M_Run();
	M_ErrorHandling();
END_IF


// Manual/Automatic mode
trigManOn(CLK := bCmdManual);
trigAutoOn(CLK := bCmdAuto);

IF (trigManOn.Q) THEN
	rManualValue := rActualValue;
	bStaManual := TRUE;
	bCmdManual := FALSE;

ELSIF (trigAutoOn.Q) THEN
	rActualValue := rAutoValue;
	bStaManual := FALSE;
	bCmdAuto := FALSE;

END_IF

// Run Manual/Automatic methods (overwrite them in inherited FB's)
IF (bStaManual) THEN
	M_ManualMode();
ELSE
	M_AutoMode();
END_IF

// Error reset
IF (bCmdReset) THEN
	bStaError := FALSE;
	bStaWarning := FALSE;
	eStaErrorID := E_ComponentErrors.OK;
	bCmdReset := FALSE;

END_IF

METHOD PROTECTED M_AutoMode : BOOL
VAR_INPUT
END_VAR

// Overwrite in inherited FB's!
;
END_METHOD

METHOD PROTECTED M_ErrorHandling : BOOL
VAR_INPUT
END_VAR

// Overwrite in inherited FB's!
;
END_METHOD

METHOD PROTECTED M_Init : BOOL
VAR_INPUT
END_VAR

// Overwrite in inherited FB's!
bInitDone := TRUE;
END_METHOD

METHOD PROTECTED M_ManualMode : BOOL
VAR_INPUT
END_VAR

// Overwrite in inherited FB's!
;
END_METHOD

METHOD PROTECTED M_Run : BOOL
VAR_INPUT
END_VAR

// Overwrite in inherited FB's!
;
END_METHOD

PROPERTY P_bEnable : BOOL
GET
P_bEnable := bCmdEnable;
END_GET
SET
bCmdEnable := P_bEnable;
END_SET
END_PROPERTY

PROPERTY PUBLIC P_bError : BOOL
GET

P_bError := bStaError;
END_GET
END_PROPERTY

PROPERTY PUBLIC P_bManualMode : BOOL
GET
P_bManualMode := bStaManual;
END_GET
SET // PUBLIC

IF (P_bManualMode AND NOT bStaManual) THEN
	bCmdAuto := FALSE;
	bCmdManual := TRUE;

ELSIF (NOT P_bManualMode AND bStaManual) THEN
	bCmdAuto := TRUE;
	bCmdManual := FALSE;
	
END_IF
END_SET
END_PROPERTY

PROPERTY PUBLIC P_bReset : BOOL
SET
bCmdReset := P_bReset;
END_SET
END_PROPERTY

PROPERTY PUBLIC P_rManualValue : LREAL
GET
P_rManualValue := rManualValue;
END_GET
SET
IF (P_bManualMode) THEN
	rManualValue := P_rManualValue;
END_IF
END_SET
END_PROPERTY

// Component name
PROPERTY PUBLIC P_sName : STRING
GET
P_sName := sName;
END_GET
SET
sName := P_sName;
END_SET
END_PROPERTY

// Tag name
PROPERTY PUBLIC P_sTag : STRING
GET
P_sTag := sTag;
END_GET
SET
sTag := P_sTag;
END_SET
END_PROPERTY

END_FUNCTION_BLOCK

// ---- ECC/Components/FB_LIN_TRAFO.TcPOU
FUNCTION_BLOCK FB_LIN_TRAFO
VAR_INPUT
	rIN			: LREAL;		(* input value*)
	rIN_MIN		: LREAL;		(* minimum input value *)
	rIN_MAX		: LREAL;		(* maximum input value *)
	rOUT_MIN	: LREAL;		(* corresponding minimum output value *)
	rOUT_MAX	: LREAL;		(* corresponding maximum output value *)
END_VAR
VAR_OUTPUT
	rOUT		: LREAL;		(* output value *)
	bERROR		: BOOL;			(* error: IN_MIN = IN_MAX or IN out of interval *)
END_VAR

VAR
	rA			: LREAL;
	rB			: LREAL;
END_VAR


IF rIN_MIN<> rIN_MAX
AND rOUT_MIN<>rOUT_MAX THEN
	(*	A=(Y2-Y1)/(X2-X1) 		*)
	rA:=(rOUT_MAX-rOUT_MIN)/(rIN_MAX-rIN_MIN);
	(* 	B=Y2-A*X2 			*)
	rB:=rOUT_MAX-rA*rIN_MAX;

	(* Y=A*X+b *)
	rOUT:=rA*rIN+rB;

	IF rOUT_MIN<rOUT_MAX THEN
		IF rOUT<rOUT_MIN THEN
			rOUT:=rOUT_MIN;
		ELSIF rOUT>rOUT_MAX THEN
			rOUT:=rOUT_MAX;
		END_IF
	ELSE
		IF rOUT>rOUT_MIN THEN
			rOUT:=rOUT_MIN;
		ELSIF rOUT<rOUT_MAX THEN
			rOUT:=rOUT_MAX;
		END_IF
	END_IF

	bERROR:=FALSE;
ELSE
	bERROR:=TRUE;
END_IF

END_FUNCTION_BLOCK

// ---- ECC/Components/F_ECat_OK.TcPOU
FUNCTION F_ECat_OK : BOOL
VAR_INPUT
	State : WORD;	// State from Ethercat module/device
END_VAR
VAR
END_VAR

// Check etherCAT state OK
F_ECat_OK := (State AND 16#0008) = 8;
IF bTestMode THEN
	F_ECat_OK := TRUE;
END_IF

END_FUNCTION

// ---- ECC/Components/FB_AO.TcPOU
FUNCTION_BLOCK FB_AO EXTENDS FB_Basic
VAR_INPUT
	rValue		: LREAL;
END_VAR
VAR_OUTPUT
END_VAR
VAR
	fbLinTrafo	: FB_LIN_TRAFO;

// HW
	{attribute 'OPC.UA.DA':='1'}
	{attribute 'OPC.UA.DA.Access' := '1'}
	{attribute 'OPC.UA.DA.Description' := 'Output I/O signal (RAW)'}
	{attribute 'OPC.UA.DA.StructuredType' := '0'}
	AnalogOutput AT %Q* : INT;	// Value to IO module
	State AT %I* : UINT := 8;	// State from Ethercat module
	AdsAdrr AT %I* : AMSADDR;	// ADS address from EtherCAT module

END_VAR
VAR PERSISTENT
	rScaleMax	: LREAL := 100;
	rScaleMin	: LREAL := -100;

END_VAR


// Run parent FB
SUPER^();

METHOD PROTECTED M_AutoMode : BOOL
VAR_INPUT
END_VAR
// Analog output automatic mode
// Executed from parent FB_Basic

rAutoValue := rValue;

IF (P_bEnable) THEN
	rActualValue := rAutoValue;
ELSE
	rActualValue := 0.0;
END_IF
END_METHOD

METHOD PROTECTED M_ErrorHandling : BOOL
VAR_INPUT
END_VAR
// Error handling
IF (bCmdEnable) THEN
	IF (NOT P_bManualMode) THEN
		// Hardware errors
		IF (NOT F_ECat_OK(State)) THEN
			// EtherCAT state
			bStaError := TRUE;
			eStaErrorID := E_ComponentErrors.HW_ECat_Not_OP;
		END_IF
	END_IF
	
ELSE
	bStaError := FALSE;
	bStaWarning := FALSE;
	eStaErrorID := E_ComponentErrors.OK;

END_IF
END_METHOD

METHOD PROTECTED M_Init : BOOL
VAR_INPUT
END_VAR
// Init

bCmdEnable := TRUE;
bInitDone := TRUE;
END_METHOD

METHOD PROTECTED M_ManualMode : BOOL
VAR_INPUT
END_VAR
// Analog Output manual mode
// Executed from parent FB_Basic

rManualValue := LIMIT(rScaleMin, rManualValue, rScaleMax);

IF (P_bEnable) THEN
	rActualValue := rManualValue;
ELSE
	rActualValue := 0.0;
END_IF
END_METHOD

METHOD PROTECTED M_Run : BOOL
VAR_INPUT
END_VAR
// Analog outputs run
// Executed from parent FB_Basic

// Update IO 

fbLinTrafo(	rIN := rActualValue,
			rIN_MIN := rScaleMin,
			rIN_MAX := rScaleMax,
			rOUT_MIN := -32767,
			rOUT_MAX := 32767,
			rOUT => ,
			bERROR =>	);

AnalogOutput := LREAL_TO_INT(fbLinTrafo.rOUT);
END_METHOD

PROPERTY PUBLIC P_rScaleMax : LREAL
GET
P_rScaleMax := rScaleMax;
END_GET
SET
rScaleMax := P_rScaleMax;
END_SET
END_PROPERTY

PROPERTY PUBLIC P_rScaleMin : LREAL
GET
P_rScaleMin := rScaleMin;
END_GET
SET
rScaleMin := P_rScaleMin;
END_SET
END_PROPERTY

END_FUNCTION_BLOCK

// ---- ECC/Components/FB_Blink.TcPOU
/// Q0 produces a High-Signal with the length OF PT on every rising edge on IN.
FUNCTION_BLOCK FB_Blink
VAR_INPUT
	IN			: BOOL;		// TRUE:run Blink, FALSE: Q = FALSE
	PT_L		: TIME;		// Time for Q = FALSE
	PT_H		: TIME;		// Time for Q = TRUE
END_VAR
VAR_OUTPUT
	Q			:BOOL;		// output variable, starting with FALSE
END_VAR
VAR
	CLOCK:TON;
END_VAR


IF (IN) THEN
	IF (Q) THEN (*high time*)
		CLOCK( IN := TRUE, PT := PT_H, Q=>, ET=> );
		IF (CLOCK.Q) THEN
			CLOCK(IN := FALSE);
			Q := FALSE;
		END_IF
	ELSE (*low time*)
		CLOCK( IN := TRUE, PT := PT_L, Q=> Q, ET=> );
		IF (CLOCK.Q) THEN
			CLOCK(IN := FALSE);
			Q := TRUE;
		END_IF;
	END_IF
ELSE
	CLOCK( IN := FALSE, PT:=, Q=>, ET=> );
	Q := FALSE;
END_IF;

END_FUNCTION_BLOCK

// ---- ECC/Components/FB_Cylinder.TcPOU
FUNCTION_BLOCK FB_Cylinder EXTENDS FB_Basic
VAR_INPUT
	eCmd			: E_Cylinder_Cmd;
END_VAR
VAR_OUTPUT
	eSta			: E_Cylinder_Sta;
END_VAR
VAR
	B1				: FB_DI;		// Activated/forward reed sensor
	B2 				: FB_DI;		// Not Activated/reverse reed sensor
	K1 				: FB_DO;		// Activate valve coil forward
	K2 				: FB_DO;		// Activate valve coil reverse
	bUseB1			: BOOL;
	bUseB2			: BOOL;
	tonB1Delay		: TON;
	tonB2Delay		: TON;
END_VAR
VAR PERSISTENT
	{attribute 'OPC.UA.DA':='1'}
	{attribute 'OPC.UA.DA.Access' := '3'}
	{attribute 'OPC.UA.DA.Description' := 'B1 sensor delay'}
	{attribute 'OPC.UA.DA.StructuredType' := '0'}
	tB1Delay		: TIME := T#5S;	// Delay forward reached (B1/K1) 
	{attribute 'OPC.UA.DA':='1'}
	{attribute 'OPC.UA.DA.Access' := '3'}
	{attribute 'OPC.UA.DA.Description' := 'B2 sensor delay'}
	{attribute 'OPC.UA.DA.StructuredType' := '0'}
	tB2Delay		: TIME := T#5S;	// Delay reverse reached (B2/K2)
END_VAR


// Run parent FB
SUPER^();

METHOD PUBLIC M_Activate : BOOL
VAR_INPUT
END_VAR
eCmd := E_Cylinder_Cmd.Cyl_Cmd_Fwd;
M_Activate := (eSta = E_Cylinder_Sta.Cyl_Sta_Fwd);
END_METHOD

METHOD PROTECTED M_AutoMode : BOOL
VAR_INPUT
END_VAR
// Digital outputs automatic mode
// Executed from parent FB_Basic

IF (eCmd = Cyl_Cmd_Fwd) THEN
	rAutoValue := 1;
ELSIF (eCmd = Cyl_Cmd_Rev) THEN
	rAutoValue := -1;
ELSE
	rAutoValue := 0;
END_IF

IF (P_bEnable) THEN
	rActualValue := rAutoValue;
ELSE
	rActualValue := 0.0;
END_IF
END_METHOD

METHOD PUBLIC M_Deactivate : BOOL
VAR_INPUT
END_VAR
eCmd := E_Cylinder_Cmd.Cyl_Cmd_Rev;
M_Deactivate := (eSta = E_Cylinder_Sta.Cyl_Sta_Rev);
END_METHOD

METHOD PROTECTED M_ErrorHandling : BOOL
VAR_INPUT
END_VAR
END_METHOD

METHOD PROTECTED M_Init : BOOL
VAR_INPUT
END_VAR

// Nothing to init
bInitDone := TRUE;
END_METHOD

METHOD PUBLIC M_IsActivated : BOOL
VAR_INPUT
END_VAR
M_IsActivated := (eSta = E_Cylinder_Sta.Cyl_Sta_Fwd);
END_METHOD

METHOD PUBLIC M_IsDeactivated : BOOL
VAR_INPUT
END_VAR
M_IsDeactivated := (eSta = E_Cylinder_Sta.Cyl_Sta_Rev);
END_METHOD

METHOD PUBLIC M_IsStopped : BOOL
VAR_INPUT
END_VAR
M_IsStopped := (eCmd = Cyl_Cmd_None);
END_METHOD

METHOD PROTECTED M_ManualMode : BOOL
VAR_INPUT
END_VAR
// Cylinder manual mode
// Executed from parent FB_Basic

// rManualValue set from e.g. HMI
// 1 => activate cylinder

rManualValue := LIMIT(-1, rManualValue, 1);

IF (P_bEnable) THEN
	rActualValue := rManualValue;
ELSE
	rActualValue := 0.0;
END_IF

B1.bValue;
B2.bValue;
END_METHOD

METHOD PROTECTED M_Run : BOOL
VAR_INPUT
END_VAR

// Feedback
B1();
B2();
IF (bUseB1 AND bUseB2 AND NOT bTestMode) THEN
	// Use both reed sensors
	tonB1Delay(IN := B1.bValue, PT := tB1Delay);
	tonB2Delay(IN := B2.bValue, PT := tB2Delay);
ELSIF (bUseB1 AND NOT bUseB2 AND NOT bTestMode) THEN
	// Only use B1 (Forward) reed sensor
	tonB1Delay(IN := B1.bValue, PT := tB1Delay);
	tonB2Delay(IN := K2.bValue, PT := tB2Delay);
ELSIF (NOT bUseB1 AND bUseB2 AND NOT bTestMode) THEN
	// Only use B2 (Reverse) reed sensor
	tonB1Delay(IN := K1.bValue, PT := tB1Delay);
	tonB2Delay(IN := B2.bValue, PT := tB2Delay);
ELSE
	// Don't use any reed sensors
	tonB1Delay(IN := K1.bValue, PT := tB1Delay);
	tonB2Delay(IN := K2.bValue, PT := tB2Delay);
END_IF

IF (tonB1Delay.Q AND NOT tonB2Delay.Q) THEN
	eSta := Cyl_Sta_Fwd;
ELSIF (tonB2Delay.Q AND NOT tonB1Delay.Q) THEN
	eSta := Cyl_Sta_Rev;
ELSIF (tonB1Delay.Q AND tonB2Delay.Q) THEN
	eSta := Cyl_Sta_Err;
ELSE
	eSta := Cyl_Sta_None;
END_IF


// Command outputs
K1.P_bEnable := P_bEnable;
K2.P_bEnable := P_bEnable;
IF (rActualValue >= 1) THEN
	K1.bValue := TRUE;
	K2.bValue := FALSE;
ELSIF (rActualValue <= -1) THEN
	K1.bValue := FALSE;
	K2.bValue := TRUE;	
ELSE
	K1.bValue := FALSE;
	K2.bValue := FALSE;	
END_IF

K1();
K2();
END_METHOD

METHOD PUBLIC M_Stop : BOOL
VAR_INPUT
END_VAR
eCmd := E_Cylinder_Cmd.Cyl_Cmd_None;
M_Stop := (NOT K1.bValue AND NOT K2.bValue);
END_METHOD

PROPERTY PUBLIC P_bUseB1 : BOOL
GET
P_bUseB1 := bUseB1;
END_GET
SET
bUseB1 := P_bUseB1;
END_SET
END_PROPERTY

PROPERTY PUBLIC P_bUseB2 : BOOL
GET
P_bUseB2 := bUseB2;
END_GET
SET
bUseB2 := P_bUseB2;
END_SET
END_PROPERTY

PROPERTY PUBLIC P_rB1Delay : REAL
GET

P_rB1Delay := (TIME_TO_REAL(tB1Delay) / 1000.0);
END_GET
SET

tB1Delay := REAL_TO_TIME(P_rB1Delay * 1000.0);
END_SET
END_PROPERTY

PROPERTY PUBLIC P_rB2Delay : REAL
GET

P_rB2Delay := (TIME_TO_REAL(tB2Delay) / 1000.0);
END_GET
SET

tB2Delay := REAL_TO_TIME(P_rB2Delay * 1000.0);
END_SET
END_PROPERTY

END_FUNCTION_BLOCK

// ---- ECC/Components/FB_DI.TcPOU
FUNCTION_BLOCK FB_DI EXTENDS FB_Basic
VAR_INPUT
END_VAR
VAR_OUTPUT
	bValue		: BOOL;
END_VAR
VAR
// HW
	{attribute 'OPC.UA.DA':='1'}
	{attribute 'OPC.UA.DA.Access' := '1'}
	{attribute 'OPC.UA.DA.Description' := 'Input I/O signal'}
	{attribute 'OPC.UA.DA.StructuredType' := '0'}
	Input AT %I* : BOOL;		// Value to IO module
	State AT %I* : WORD := 8;	// State from Ethercat module

END_VAR
VAR PERSISTENT
	bUseLoLo	: BOOL;
	bUseLo		: BOOL;
	bUseHi		: BOOL;
	bUseHiHi	: BOOL;

END_VAR


// Run parent FB
SUPER^();

METHOD PROTECTED M_AutoMode : BOOL
VAR_INPUT
END_VAR
// Analog inputs automatic mode
// Executed from parent FB_Basic

IF (P_bEnable) THEN
	rActualValue := rAutoValue;
ELSE
	rActualValue := 0;
END_IF

bValue := LREAL_TO_BOOL(rActualValue);
END_METHOD

METHOD PROTECTED M_ErrorHandling : BOOL
VAR_INPUT
END_VAR
// Error handling
IF (bCmdEnable) THEN
	IF (NOT P_bManualMode) THEN
		// Hardware errors
		IF (NOT F_ECat_OK(State)) THEN
			// EtherCAT state
			bStaError := TRUE;
			eStaErrorID := E_ComponentErrors.HW_ECat_Not_OP;
		END_IF
	END_IF

	// Software errors
	IF (bUseHiHi AND bValue) THEN
		bStaError := TRUE;
		eStaErrorID := E_ComponentErrors.SW_HiHi;
	END_IF
	IF (bUseHi AND bValue) THEN
		bStaWarning := TRUE;
		eStaErrorID := E_ComponentErrors.SW_Hi;
	END_IF
	IF (bUseLoLo AND NOT bValue) THEN
		bStaError := TRUE;
		eStaErrorID := E_ComponentErrors.SW_LoLo;
	END_IF
	IF (bUseLo AND NOT bValue) THEN
		bStaWarning := TRUE;
		eStaErrorID := E_ComponentErrors.SW_Lo;
	END_IF	
ELSE
	bStaError := FALSE;
	bStaWarning := FALSE;
	eStaErrorID := E_ComponentErrors.OK;

END_IF
END_METHOD

METHOD PROTECTED M_Init : BOOL
VAR_INPUT
END_VAR
// Init

bCmdEnable := TRUE;
bInitDone := TRUE;
END_METHOD

METHOD PROTECTED M_ManualMode : BOOL
VAR_INPUT
END_VAR
// Analog inputs manual mode
// Executed from parent FB_Basic

rManualValue := LIMIT(0, rManualValue, 1);

IF (P_bEnable) THEN
	rActualValue := rManualValue;
ELSE
	rActualValue := 0.0;
END_IF

bValue := LREAL_TO_BOOL(rActualValue);
END_METHOD

METHOD PROTECTED M_Run : BOOL
VAR_INPUT
END_VAR
// Analog inputs run
// Executed from parent FB_Basic

// Update IO

rAutoValue := BOOL_TO_LREAL(Input);
END_METHOD

END_FUNCTION_BLOCK

// ---- ECC/Components/FB_DO.TcPOU
FUNCTION_BLOCK FB_DO EXTENDS FB_Basic
VAR_INPUT
	bValue		: BOOL;

END_VAR
VAR_OUTPUT
END_VAR
VAR
// HW
	{attribute 'OPC.UA.DA':='1'}
	{attribute 'OPC.UA.DA.Access' := '1'}
	{attribute 'OPC.UA.DA.Description' := 'Output I/O signal'}
	{attribute 'OPC.UA.DA.StructuredType' := '0'}
	Output AT %Q* : BOOL;		// Value to IO module
	State AT %I* : WORD := 8;	// State from Ethercat module

END_VAR


// Run parent FB
SUPER^();

METHOD PROTECTED M_AutoMode : BOOL
VAR_INPUT
END_VAR
// Digital outputs automatic mode
// Executed from parent FB_Basic

rAutoValue := BOOL_TO_LREAL(bValue);

IF (P_bEnable) THEN
	rActualValue := rAutoValue;
ELSE
	rActualValue := 0.0;
END_IF
END_METHOD

METHOD PROTECTED M_ErrorHandling : BOOL
VAR_INPUT
END_VAR
// Error handling
IF (bCmdEnable) THEN
	IF (NOT P_bManualMode) THEN
		// Hardware errors
		IF (NOT F_ECat_OK(State)) THEN
			// EtherCAT state
			bStaError := TRUE;
			eStaErrorID := E_ComponentErrors.HW_ECat_Not_OP;
		END_IF
	END_IF
	
ELSE
	bStaError := FALSE;
	bStaWarning := FALSE;
	eStaErrorID := E_ComponentErrors.OK;

END_IF
END_METHOD

METHOD PROTECTED M_Init : BOOL
VAR_INPUT
END_VAR
// Init

bCmdEnable := TRUE;
bInitDone := TRUE;
END_METHOD

METHOD PROTECTED M_ManualMode : BOOL
VAR_INPUT
END_VAR
// Digital outputs manual mode
// Executed from parent FB_Basic

rManualValue := LIMIT(0, rManualValue, 1);

IF (P_bEnable) THEN
	rActualValue := rManualValue;
ELSE
	rActualValue := 0.0;
END_IF
END_METHOD

METHOD PROTECTED M_Run : BOOL
VAR_INPUT
END_VAR
// Analog inputs run
// Executed from parent FB_Basic

// Update IO 

Output := LREAL_TO_BOOL(rActualValue);
END_METHOD

END_FUNCTION_BLOCK

// ---- ECC/Components/TwinSAFE/FB_TwinSAFE_Group.TcPOU
FUNCTION_BLOCK FB_TwinSAFE_Group EXTENDS FB_Basic
VAR_INPUT
END_VAR
VAR_OUTPUT
END_VAR
VAR
	State AT %I* : UINT := 8;	// State from Ethercat module
	// Map to TwinSAFE group State (Remember to activate Map State in TwinSAFE group infodata)
	{attribute 'OPC.UA.DA':='1'}
	{attribute 'OPC.UA.DA.Access' := '1'}
	{attribute 'OPC.UA.DA.Description' := 'TwinSAFE group state'}
	{attribute 'OPC.UA.DA.StructuredType' := '0'}
	GroupState AT %I*			: E_TwinSAFE_Group_State;
	// Map to TwinSAFE group State (Remember to activate Map Diag in TwinSAFE group infodata)
	{attribute 'OPC.UA.DA':='1'}
	{attribute 'OPC.UA.DA.Access' := '1'}
	{attribute 'OPC.UA.DA.Description' := 'TwinSAFE group diag'}
	{attribute 'OPC.UA.DA.StructuredType' := '0'}
	GroupDiag AT %I*			: E_TwinSAFE_Group_Diag;
	// Map to TwinSAFE FSLOGICS inputs
	SafeLogicState AT %I*		: E_TwinSAFE_Logic_State;
	// Map to TwinSAFE FSLOGICS inputs
	CycleCounter AT %I*			: USINT;
	// Map to ErrorAcknowledgement in TwinSAFE group
	{attribute 'OPC.UA.DA':='1'}
	{attribute 'OPC.UA.DA.Access' := '1'}
	{attribute 'OPC.UA.DA.Description' := 'TwinSAFE group acknowledgment'}
	{attribute 'OPC.UA.DA.StructuredType' := '0'}
	ErrorAcknowledgement AT %Q*	: BOOL;
	// Map to Run in TwinSAFE group
	{attribute 'OPC.UA.DA':='1'}
	{attribute 'OPC.UA.DA.Access' := '1'}
	{attribute 'OPC.UA.DA.Description' := 'TwinSAFE group run'}
	{attribute 'OPC.UA.DA.StructuredType' := '0'}
	Run AT %Q*					: BOOL;
	tpReset: TP;
END_VAR


// Run parent FB
SUPER^();

METHOD PROTECTED M_ErrorHandling : BOOL
VAR_INPUT
END_VAR
// Error handling
IF (bCmdEnable) THEN
	IF (State < 8) THEN
		// EtherCAT state
		bStaError := TRUE;
		eStaErrorID := E_ComponentErrors.HW_ECat_Not_OP;
	ELSE
		CASE GroupState OF
			E_TwinSAFE_Group_State.RUN:
				bStaError := FALSE;
				eStaErrorID := E_ComponentErrors.OK;
			
			E_TwinSAFE_Group_State.STOP:
				bStaError := TRUE;
				eStaErrorID := E_ComponentErrors.TS_Stop;
			
			E_TwinSAFE_Group_State.ERROR:
				bStaError := TRUE;
				CASE GroupDiag OF
					E_TwinSAFE_Group_Diag.NO_ERROR:
						eStaErrorID := E_ComponentErrors.TS_Error;
						
					E_TwinSAFE_Group_Diag.FBERROR:
						eStaErrorID := E_ComponentErrors.TS_FBError;
	
					E_TwinSAFE_Group_Diag.COMERROR:
						eStaErrorID := E_ComponentErrors.TS_ComError;
	
					E_TwinSAFE_Group_Diag.MODULEERROR:
						eStaErrorID := E_ComponentErrors.TS_ModuleError;
	
					E_TwinSAFE_Group_Diag.CMPERROR:
						eStaErrorID := E_ComponentErrors.TS_CMPError;
	
					E_TwinSAFE_Group_Diag.DEACTIVATEERROR:
						eStaErrorID := E_ComponentErrors.TS_DeactivateError;
	
					E_TwinSAFE_Group_Diag.RESTARTERROR:
						eStaErrorID := E_ComponentErrors.TS_RestartError;
	
				END_CASE
	
			E_TwinSAFE_Group_State.START:
				bStaError := FALSE;
				eStaErrorID := E_ComponentErrors.OK;
			
			E_TwinSAFE_Group_State.STOPERROR:
				bStaError := TRUE;
				eStaErrorID := E_ComponentErrors.TS_StopError;
	
			E_TwinSAFE_Group_State.DEACTIVE:
				bStaError := TRUE;
				eStaErrorID := E_ComponentErrors.TS_Deactivated;
	
			E_TwinSAFE_Group_State.WAITCOMERROR:
				bStaError := TRUE;
				eStaErrorID := E_ComponentErrors.TS_WaitCommError;
	
		END_CASE
	END_IF

ELSE
	bStaError := FALSE;
	bStaWarning := FALSE;
	eStaErrorID := E_ComponentErrors.OK;

END_IF
END_METHOD

METHOD PROTECTED M_Init : BOOL
VAR_INPUT
END_VAR
// Init

bCmdEnable := TRUE;
bInitDone := TRUE;
END_METHOD

METHOD PROTECTED M_Run : BOOL
VAR_INPUT
END_VAR
// Analog outputs run
// Executed from parent FB_Basic

// Enable TwinSAFE group
IF (P_bEnable) THEN
	Run := TRUE;
ELSE
	Run := FALSE;
END_IF

// Reset TwinSAFE group
tpReset(IN := bCmdReset, PT := T#500MS, Q => ErrorAcknowledgement);
END_METHOD

END_FUNCTION_BLOCK

// ---- ECC/Tools/FB_OPCUA_Client_Basic.TcPOU
FUNCTION_BLOCK FB_OPCUA_Client_Basic
VAR_INPUT
	bExecute 			: BOOL;	// Start reading
	sVarName			: STRING(MAX_STRING_LENGTH); // Variable to read from OPC UA server
	eUAIdentifierType	: Tc3_PLCopen_OpcUa.E_UAIdentifierType := Tc3_PLCopen_OpcUa.eUAIdentifierType_Numeric;
END_VAR
VAR_OUTPUT
	bDone		: BOOL;		// TRUE when completed without errors
	bBusy		: BOOL;		// TRUE when working
	bError		: BOOL;		// TRUE if error
	nErrorID	: DWORD;	// Error ID from OPC comm. FB's
END_VAR
VAR
	eState					: E_OPCUA_Client_Seq;
	(* Declarations for UA_Connect *)
	fbUA_Connect			: Tc3_PLCopen_OpcUa.UA_Connect;
	SessionConnectInfo		: Tc3_PLCopen_OpcUa.ST_UASessionConnectInfo;
	nConnectionHdl			: DWORD;
	(* Declarations for UA_GetNamespaceIndex *)
	fbUA_GetNamespaceIndex 	: Tc3_PLCopen_OpcUa.UA_GetNamespaceIndex;
	nNamespaceIndex			: UINT;
	(* Declarations for UA_NodeGetHandle *)
	fbUA_NodeGetHandle		: Tc3_PLCopen_OpcUa.UA_NodeGetHandle;
	NodeID					: Tc3_PLCopen_OpcUa.ST_UANodeID;
	nNodeHdl				: DWORD;
	(* Declarations for UA_NodeReleaseHandle *)
	fbUA_NodeReleaseHandle	: Tc3_PLCopen_OpcUa.UA_NodeReleaseHandle;
	(* Declarations for UA_Disconnect *)
	fbUA_Disconnect			: Tc3_PLCopen_OpcUa.UA_Disconnect;
END_VAR
VAR PERSISTENT
	sOpcUaServerUrl		: STRING(MAX_STRING_LENGTH) := 'opc.tcp://localhost:4840';
	sNamespaceUri		: STRING(MAX_STRING_LENGTH) := 'urn:BeckhoffAutomation:Ua:PLC1'; // TF6100 setup version 4.x default
END_VAR

METHOD PROTECTED M_CloseSession : E_Method
VAR_INPUT
END_VAR

	fbUA_Disconnect(Execute := TRUE,
					ConnectionHdl := nConnectionHdl	);

	IF (fbUA_Disconnect.Busy) THEN
		M_CloseSession := E_Method.Busy;
	ELSIF (fbUA_Disconnect.Error) THEN
		fbUA_Disconnect(Execute := FALSE);
		bError := TRUE;
		nErrorID := fbUA_Disconnect.ErrorID;
		nConnectionHdl := 0;
		M_CloseSession := E_Method.Error;
	ELSIF (fbUA_Disconnect.Done) THEN		
		fbUA_Disconnect(Execute := FALSE);
		IF (NOT bError) THEN 
			bDone := TRUE;
		END_IF
		M_CloseSession := E_Method.Done;
	ELSE
		M_CloseSession := E_Method.Idle;			
	END_IF
END_METHOD

/// Get namespace index -  1: Busy, 2: Done, 5: Error
METHOD PROTECTED M_GetNameSpace : E_Method
VAR_INPUT
END_VAR
	fbUA_GetNamespaceIndex(	Execute := TRUE,
							ConnectionHdl := nConnectionHdl,
							NamespaceUri := sNamespaceUri,
							NamespaceIndex => nNamespaceIndex	);

	IF (fbUA_GetNamespaceIndex.Busy) THEN
		M_GetNameSpace := E_Method.Busy;			
	ELSIF (fbUA_GetNamespaceIndex.Error) THEN
		// Get namespace index failed
		fbUA_GetNamespaceIndex(Execute := FALSE);
		bError := TRUE;
		nErrorID := fbUA_GetNamespaceIndex.ErrorID;
		M_GetNameSpace := E_Method.Error;
	ELSIF (fbUA_GetNamespaceIndex.Done) THEN
		// Namespace index obtained
		fbUA_GetNamespaceIndex(Execute := FALSE);
		M_GetNameSpace := E_Method.Done;
	ELSE
		M_GetNameSpace := E_Method.Idle;			
	END_IF
END_METHOD

/// Open session -  1: Busy, 2: Done, 5: Error
METHOD PROTECTED M_GetNode : E_Method
VAR_INPUT
END_VAR

	NodeID.eIdentifierType := eUAIdentifierType;
	NodeID.nNamespaceIndex := nNamespaceIndex;
	NodeID.sIdentifier := sVarName;
	fbUA_NodeGetHandle(	Execute := TRUE,
						ConnectionHdl := nConnectionHdl,
						NodeID := NodeID,
						NodeHdl => nNodeHdl	);

	IF (fbUA_NodeGetHandle.Busy) THEN
		// Obtaining handle
		M_GetNode := E_Method.Busy;
	ELSIF (fbUA_NodeGetHandle.Error) THEN
		// Error ontaining handle
		fbUA_NodeGetHandle(Execute := FALSE);
		bError := TRUE;
		nErrorID := fbUA_NodeGetHandle.ErrorID;
		M_GetNode := E_Method.Error;
	ELSIF (fbUA_NodeGetHandle.Done) THEN
		// Handle obtained
		fbUA_NodeGetHandle(Execute := FALSE);
		M_GetNode := E_Method.Done;
	ELSE
		M_GetNode := E_Method.Idle;			
	END_IF
END_METHOD

METHOD PROTECTED M_Init : E_Method
VAR_INPUT
END_VAR
	bError := FALSE;
	nErrorID := 0;
	bBusy := TRUE;

	SessionConnectInfo.tConnectTimeout := T#1M;
	SessionConnectInfo.tSessionTimeout := T#1M;
	SessionConnectInfo.sApplicationName := '';
	SessionConnectInfo.eSecurityMode := eUASecurityMsgMode_None;
	SessionConnectInfo.eSecurityPolicyUri := eUASecurityPolicy_None;
	SessionConnectInfo.eTransportProfileUri := eUATransportProfileUri_UATcp;

	M_Init := E_Method.Done;
END_METHOD

/// Open session -  1: Busy, 2: Done, 5: Error
METHOD PROTECTED M_OpenSession : E_Method
VAR_INPUT
END_VAR
	fbUA_Connect(	Execute := TRUE,
					ServerURL := sOpcUaServerUrl,
					SessionConnectInfo := SessionConnectInfo,
					Timeout := T#5S,
					ConnectionHdl => nConnectionHdl	);

	IF (fbUA_Connect.Busy) THEN
		// Session opening
		M_OpenSession := E_Method.Busy;
	ELSIF (fbUA_Connect.Error) THEN
		// Error opening session
		fbUA_Connect(Execute := FALSE);
		bError := TRUE;
		nErrorID := fbUA_Connect.ErrorID;
		nConnectionHdl := 0;
		M_OpenSession := E_Method.Error;
	ELSIF (fbUA_Connect.Done) THEN
		// session opened
		fbUA_Connect(Execute := FALSE);
		M_OpenSession := E_Method.Done;
	ELSE
		M_OpenSession := E_Method.Idle;			
	END_IF
END_METHOD

METHOD PROTECTED M_ReleaseNode : E_Method
VAR_INPUT
END_VAR

	fbUA_NodeReleaseHandle(	Execute := TRUE,
							ConnectionHdl := nConnectionHdl,
							NodeHdl := nNodeHdl	);

	IF (fbUA_NodeReleaseHandle.Busy) THEN
		// Working
		M_ReleaseNode := E_Method.Busy;
	ELSIF (fbUA_NodeReleaseHandle.Error) THEN
		// Error releasing node handle
		fbUA_NodeReleaseHandle(Execute := FALSE);
		bError := TRUE;
		nErrorID := fbUA_NodeReleaseHandle.ErrorID;
		M_ReleaseNode := E_Method.Error;		
	ELSIF (fbUA_NodeReleaseHandle.Done) THEN
		// Node handle released
		fbUA_NodeReleaseHandle(Execute := FALSE);
		M_ReleaseNode := E_Method.Done;
	ELSE
		M_ReleaseNode := E_Method.Idle;			
	END_IF
END_METHOD

PROPERTY PUBLIC P_sNamespaceUri : STRING(MAX_STRING_LENGTH)
GET
P_sNamespaceUri := sNamespaceUri;
END_GET
SET
sNamespaceUri := P_sNamespaceUri;
END_SET
END_PROPERTY

PROPERTY PUBLIC P_sOpcUaServerUrl : STRING(MAX_STRING_LENGTH)
GET
P_sOpcUaServerUrl := sOpcUaServerUrl;
END_GET
SET
sOpcUaServerUrl := P_sOpcUaServerUrl;
END_SET
END_PROPERTY

END_FUNCTION_BLOCK

// ---- ECC/Tools/FB_OPCUA_Client_CallMethod.TcPOU
FUNCTION_BLOCK FB_OPCUA_Client_CallMethod EXTENDS FB_OPCUA_Client_Basic
VAR_INPUT
	iTargetSize	: UDINT;	// Size of local target variable
	pTarget		: pVoid;	// Address of local target variable
	sObjectName	: STRING(MAX_STRING_LENGTH);	// program/FB name
	sMethodName	: STRING(MAX_STRING_LENGTH);	// Method name
	iNoOfInArgs	: UINT;		// Number of input arguments
	iInputArgs	: ARRAY [0..10] OF INT;			// input Arguments for method
END_VAR
VAR_OUTPUT
END_VAR
VAR
	(* Declarations for UA_MethodGetHandle *)
	fbUA_MethodGetHandle: UA_MethodGetHandle;
	ObjectNodeID: ST_UANodeID;
	MethodNodeID: ST_UANodeID;
	nMethodHdl: DWORD;
	(* Declarations for UA_MethodCall *)
	fbUA_MethodCall: UA_MethodCall;
	nAdrWriteData: PVOID;
	cbWriteData: UDINT; // calculated automatically by M_Init()
	InputArguments: ARRAY[1..10] OF ST_UAMethodArgInfo; // change according to input parameters - M_Mul has 2 input parameters 
	stOutputArgInfo: ARRAY[1..1] OF ST_UAMethodArgInfo; // change according to output parameters - M_Mul has 1 output parameters
	stOutputArgInfoAndData: ST_OutputArgInfoAndData_Recipe;
	nInputData: ARRAY[1..20] OF BYTE; // numberIn1(INT16)(2) + numberIn2(INT16)(2)
	nOffset: UDINT; // calculated by M_Init()
	nArg: INT; // used by M_Init()
	(* Declarations for UA_MethodReleaseHandle *)
	fbUA_MethodReleaseHandle: UA_MethodReleaseHandle;
	
	nNumberOfInputArguments: DINT := 2; // change to number of input parameters - M_Mul has 2 input parameters
	nInputArgSize: INT := 20; // numberIn1(INT16)(2) + numberIn2(INT16)(2)
	bHandleInited : BOOL;
END_VAR
VAR CONSTANT
//	nInputArgSize: INT := 4; // numberIn1(INT16)(2) + numberIn2(INT16)(2)
//	nNumberOfInputArguments: DINT := 2; // change to number of input parameters - M_Mul has 2 input parameters
	nNumberOfOutputArguments: DINT := 1; // change to number of output parameters - M_Mul has 1 output parameters
END_VAR

CASE eState OF
	E_OPCUA_Client_Seq.Idle:
		IF (bExecute) THEN
			M_Init();
			eState := E_OPCUA_Client_Seq.CheckData;
		END_IF

	E_OPCUA_Client_Seq.CheckData:
		IF ((sMethodName <> '') AND (sObjectName <> '') AND (pTarget <> 0) AND (iTargetSize > 0)) THEN
			eState := E_OPCUA_Client_Seq.OpenSession;
		ELSE
			bError := TRUE;
			bBusy := FALSE;
			eState := E_OPCUA_Client_Seq.Done;
		END_IF

	E_OPCUA_Client_Seq.OpenSession:
		CASE M_OpenSession() OF
			E_Method.Done:	// Done
				eState := E_OPCUA_Client_Seq.GetNameSpace;
			E_Method.Error:	// Error
				eState := E_OPCUA_Client_Seq.Done;
		END_CASE

	E_OPCUA_Client_Seq.GetNameSpace:
		CASE M_GetNameSpace() OF
			E_Method.Done:	// Done
				eState := E_OPCUA_Client_Seq.GetMethod;
			E_Method.Error:	// Error
				eState := E_OPCUA_Client_Seq.CloseSession;			
		END_CASE

	E_OPCUA_Client_Seq.GetMethod:
		CASE M_GetMethodHandle() OF
			E_Method.Done:	// Done
				eState := E_OPCUA_Client_Seq.CallMethod;
			E_Method.Error:	// Error
				eState := E_OPCUA_Client_Seq.ReleaseMethod;
		END_CASE
		
	E_OPCUA_Client_Seq.CallMethod:
		CASE M_CallMethod() OF
			E_Method.Done:	// Done
				MEMCPY(	pTarget, ADR(stOutputArgInfoAndData.stRecipe), iTargetSize);
				eState := E_OPCUA_Client_Seq.ReleaseMethod;
			E_Method.Error:	// Error
				eState := E_OPCUA_Client_Seq.ReleaseMethod;
		END_CASE

	E_OPCUA_Client_Seq.ReleaseMethod:
		CASE M_ReleaseMethodHandle() OF
			E_Method.Done:	// Done
				eState := E_OPCUA_Client_Seq.CloseSession;
			E_Method.Error:	// Error
				eState := E_OPCUA_Client_Seq.CloseSession;
		END_CASE

	E_OPCUA_Client_Seq.CloseSession:
		CASE M_CloseSession() OF
			E_Method.Done:	// Done
				eState := E_OPCUA_Client_Seq.Done;
			E_Method.Error:	// Error
				eState := E_OPCUA_Client_Seq.Done;
		END_CASE
		
	E_OPCUA_Client_Seq.Done:
		bBusy := FALSE;
		IF (NOT bExecute) THEN
			bDone := FALSE;
			bError := FALSE;
			eState := E_OPCUA_Client_Seq.Idle;
		END_IF

	ELSE
		eState := E_OPCUA_Client_Seq.Idle;

END_CASE

METHOD PROTECTED M_CallMethod : E_Method
VAR_INPUT
END_VAR

	stOutputArgInfo[1].nLenData := SIZEOF(stOutputArgInfoAndData.stRecipe);
(*	stOutputArgInfo[1].ArrayDimensions[1] := 0;
	stOutputArgInfo[1].DataType := Tc3_PLCopen_OpcUa.eUAType_Variant;
	stOutputArgInfo[1].ValueRank := -1;
	stOutputArgInfo[1].nLenData := iTargetSize;
	stOutputArgInfoAndData.nNumberOfOutputArguments := 1;
	stOutputArgInfoAndData.stOutputArgInfo[1] := stOutputArgInfo[1];
*)
	fbUA_MethodCall(Execute := TRUE,
					ConnectionHdl := nConnectionHdl,
					MethodHdl := nMethodHdl,
					nNumberOfInputArguments := nNumberOfInputArguments,	
					pInputArgInfo := ADR(InputArguments),
					cbInputArgInfo := SIZEOF(InputArguments[1]) * nNumberOfInputArguments,
					pInputArgData := ADR(nInputData),
					cbInputArgData := cbWriteData,
					pInputWriteData := 0,
					cbInputWriteData := 0,
					nNumberOfOutputArguments := nNumberOfOutputArguments,
					pOutputArgInfo := ADR(stOutputArgInfo),
					cbOutputArgInfo := SIZEOF(stOutputArgInfo),
					pOutputArgInfoAndData := ADR(stOutputArgInfoAndData),
					cbOutputArgInfoAndData := SIZEOF(stOutputArgInfoAndData)	);
	
	IF (fbUA_MethodCall.Busy) THEN
		M_CallMethod := E_Method.Busy;
	ELSIF (fbUA_MethodCall.Error) THEN
		fbUA_MethodCall(Execute := FALSE);
		bError := TRUE;
		nErrorID := fbUA_MethodCall.ErrorID;
		M_CallMethod := E_Method.Error;
	ELSIF (fbUA_MethodCall.Done) THEN
		fbUA_MethodCall(Execute := FALSE);
		M_CallMethod := E_Method.Done;
	ELSE
		M_CallMethod := E_Method.Idle;
	END_IF
END_METHOD

METHOD PROTECTED M_GetMethodHandle : E_Method
VAR_INPUT
END_VAR
VAR
	iCnt : UINT;
	iMaxCnt : UINT;
END_VAR

IF (NOT bHandleInited) THEN
	ObjectNodeID.eIdentifierType := eUAIdentifierType_String;
	ObjectNodeID.nNamespaceIndex := nNamespaceIndex;
	ObjectNodeID.sIdentifier	 := sObjectName;

	MethodNodeID.eIdentifierType := eUAIdentifierType_String;
	MethodNodeID.nNamespaceIndex := nNamespaceIndex;
	MethodNodeID.sIdentifier	 := CONCAT(sObjectName, CONCAT('#', sMethodName));

	// Clear memory
	MEMSET(ADR(InputArguments), 0, SIZEOF(InputArguments));
	MEMSET(ADR(nInputData), 0, SIZEOF(nInputData));

	// Input arguments
	nOffset := 0;
	iMaxCnt := MIN(10, iNoOfInArgs);
	nNumberOfInputArguments := iMaxCnt;
	IF (iMaxCnt > 0) THEN
		FOR iCnt := 0 TO (iMaxCnt-1) BY 1 DO
			InputArguments[iCnt+1].DataType := Tc3_PLCopen_OpcUa.eUAType_Int16;
			InputArguments[iCnt+1].ValueRank := -1; 							(* Scalar = -1 or Array *)
			InputArguments[iCnt+1].ArrayDimensions[1] := 0; 					(* Number of Dimension in case its an array *)
			InputArguments[iCnt+1].nLenData := SIZEOF(iInputArgs[iCnt]);		(* Length if its a STRING *)
			IF (nOffset + SIZEOF(iInputArgs[iCnt]) > nInputArgSize) THEN 
				M_GetMethodHandle := E_Method.Error;
				RETURN;
			ELSE
				MEMCPY(ADR(nInputData)+nOffset,ADR(iInputArgs[iCnt]),SIZEOF(iInputArgs[iCnt]));	(* VALUE in BYTES FORM *)
				nOffset := nOffset + SIZEOF(iInputArgs[iCnt]);
			END_IF		
		END_FOR
	END_IF
	cbWriteData := nOffset;
	bHandleInited := TRUE;
END_IF

	// Get method handle	
	fbUA_MethodGetHandle(	Execute := TRUE,
							ConnectionHdl := nConnectionHdl,
							ObjectNodeID := ObjectNodeID,
							MethodNodeID := MethodNodeID,
							MethodHdl => nMethodHdl	);
	IF (fbUA_MethodGetHandle.Busy) THEN
		M_GetMethodHandle := E_Method.Busy;
	ELSIF (fbUA_MethodGetHandle.Error) THEN
		fbUA_MethodGetHandle(Execute := FALSE);
		bError := TRUE;
		nErrorID := fbUA_MethodGetHandle.ErrorID;
		M_GetMethodHandle := E_Method.Error;
	ELSIF (fbUA_MethodGetHandle.Done) THEN
		fbUA_MethodGetHandle(Execute := FALSE);
		M_GetMethodHandle := E_Method.Done;
	ELSE
		M_GetMethodHandle := E_Method.Idle;		
	END_IF
END_METHOD

METHOD PROTECTED M_Init : E_Method
VAR_INPUT
END_VAR
	
	SUPER^.M_Init();
	
	bHandleInited := FALSE;

	M_Init := E_Method.Done;
END_METHOD

METHOD PROTECTED M_ReleaseMethodHandle : E_Method
VAR_INPUT
END_VAR

	fbUA_MethodReleaseHandle(	Execute			:= TRUE,
								ConnectionHdl	:= nConnectionHdl,
								MethodHdl		:= nMethodHdl	);

	IF (fbUA_MethodReleaseHandle.Busy) THEN
		// Working
		M_ReleaseMethodHandle := E_Method.Busy;
	ELSIF (fbUA_MethodReleaseHandle.Error) THEN
		// Error releasing node handle
		fbUA_MethodReleaseHandle(Execute := FALSE);
		bError := TRUE;
		nErrorID := fbUA_MethodReleaseHandle.ErrorID;
		M_ReleaseMethodHandle := E_Method.Error;		
	ELSIF (fbUA_MethodReleaseHandle.Done) THEN
		// Node handle released
		fbUA_MethodReleaseHandle(Execute := FALSE);
		M_ReleaseMethodHandle := E_Method.Done;
	ELSE
		M_ReleaseMethodHandle := E_Method.Idle;			
	END_IF
END_METHOD

END_FUNCTION_BLOCK

// ---- ECC/Tools/FB_OPCUA_Client_ReadVar.TcPOU
FUNCTION_BLOCK FB_OPCUA_Client_ReadVar EXTENDS FB_OPCUA_Client_Basic
VAR_INPUT
	iTargetSize	: UDINT;	// Size of local target variable
	pTarget		: pVoid;	// Address of local target variable
END_VAR
VAR_OUTPUT
END_VAR
VAR
	(* Declarations for UA_Read *)
	fbUA_Read				: UA_Read;
	stIndexRange			: ARRAY [1..nMaxIndexRange] OF ST_UAIndexRange;
	nIndexRangeCount		: UINT;
	stNodeAddInfo			: ST_UANodeAdditionalInfo;
	cbDataRead				: UDINT;
END_VAR
VAR PERSISTENT
END_VAR

CASE eState OF
	E_OPCUA_Client_Seq.Idle:
		IF (bExecute) THEN
			M_Init();
			eState := E_OPCUA_Client_Seq.CheckData;
		END_IF

	E_OPCUA_Client_Seq.CheckData:
		IF ((pTarget <> 0) AND (iTargetSize > 1)) THEN
			eState := E_OPCUA_Client_Seq.OpenSession;
		ELSE
			bError := TRUE;
			bBusy := FALSE;
			eState := E_OPCUA_Client_Seq.Done;
		END_IF

	E_OPCUA_Client_Seq.OpenSession:
		CASE M_OpenSession() OF
			E_Method.Done:	// Done
				eState := E_OPCUA_Client_Seq.GetNameSpace;
			E_Method.Error:	// Error
				eState := E_OPCUA_Client_Seq.Idle;			
		END_CASE

	E_OPCUA_Client_Seq.GetNameSpace:
		CASE M_GetNameSpace() OF
			E_Method.Done:	// Done
				eState := E_OPCUA_Client_Seq.GetNode;
			E_Method.Error:	// Error
				eState := E_OPCUA_Client_Seq.CloseSession;			
		END_CASE


	E_OPCUA_Client_Seq.GetNode:
		CASE M_GetNode() OF
			E_Method.Done:	// Done
				eState := E_OPCUA_Client_Seq.Read;
			E_Method.Error:	// Error
				eState := E_OPCUA_Client_Seq.CloseSession;			
		END_CASE


	E_OPCUA_Client_Seq.Read:
		CASE M_ReadVar() OF
			E_Method.Done:	// Done
				eState := E_OPCUA_Client_Seq.ReleaseNode;
			E_Method.Error:	// Error
				eState := E_OPCUA_Client_Seq.ReleaseNode;
		END_CASE

	E_OPCUA_Client_Seq.ReleaseNode:
		CASE M_ReleaseNode() OF
			E_Method.Done:	// Done
				eState := E_OPCUA_Client_Seq.CloseSession;
			E_Method.Error:	// Error
				eState := E_OPCUA_Client_Seq.CloseSession;
		END_CASE

	E_OPCUA_Client_Seq.CloseSession:
		CASE M_CloseSession() OF
			E_Method.Done:	// Done
				eState := E_OPCUA_Client_Seq.Done;
			E_Method.Error:	// Error
				eState := E_OPCUA_Client_Seq.Done;
		END_CASE
		
	E_OPCUA_Client_Seq.Done:
		bBusy := FALSE;
		IF (NOT bExecute) THEN
			bDone := FALSE;
			bError := FALSE;
			eState := E_OPCUA_Client_Seq.Idle;
		END_IF

	ELSE
		eState := E_OPCUA_Client_Seq.Idle;

END_CASE

METHOD PROTECTED M_Init : E_Method
VAR_INPUT
END_VAR
	
	SUPER^.M_Init();	

	stNodeAddInfo.nIndexRangeCount := nIndexRangeCount;
	stNodeAddInfo.stIndexRange := stIndexRange;

	M_Init := E_Method.Done;
END_METHOD

METHOD PROTECTED M_ReadVar : E_Method
VAR_INPUT
END_VAR

	fbUA_Read(	Execute := TRUE,
				ConnectionHdl := nConnectionHdl,
				NodeHdl := nNodeHdl,
				cbData := iTargetSize,
				stNodeAddInfo := stNodeAddInfo,
				pVariable := pTarget	);

	IF (fbUA_Read.Busy) THEN
		// Reading
		M_ReadVar := E_Method.Busy;
	ELSIF (fbUA_Read.Error) THEN
		// Error reading
		fbUA_Read(Execute := FALSE);
		bError := TRUE;
		nErrorID := fbUA_Read.ErrorID;
		M_ReadVar := E_Method.Error;
	ELSIF (fbUA_Read.Done) THEN
		// Data read OK
		fbUA_Read(Execute := FALSE);
		M_ReadVar := E_Method.Done;
	ELSE
		M_ReadVar := E_Method.Idle;			
	END_IF
END_METHOD

END_FUNCTION_BLOCK

// ---- ECC/Tools/FB_OPCUA_GetRecipe.TcPOU
FUNCTION_BLOCK FB_OPCUA_GetRecipe
VAR_INPUT
END_VAR
VAR_OUTPUT
END_VAR
VAR
END_VAR

END_FUNCTION_BLOCK

// ---- ECC/Tools/FB_OPCUA_ReadVar_BAK.TcPOU
FUNCTION_BLOCK FB_OPCUA_ReadVar_BAK
VAR_INPUT
	bExecute 	: BOOL;		// Start reading
	sVarName	: STRING(MAX_STRING_LENGTH); // Variable to read from OPC UA server
	iTargetSize	: UDINT;	// Size of local target variable
	pTarget		: pVoid;	// Address of local target variable
END_VAR
VAR_OUTPUT
	bDone		: BOOL;		// TRUE when completed without errors
	bBusy		: BOOL;		// TRUE when working
	bError		: BOOL;		// TRUE if error
	nErrorID	: DWORD;	// Error ID from OPC comm. FB's
END_VAR
VAR
	eState					: E_OPCUA_Client_Seq;
	(* Declarations for UA_Connect *)
	fbUA_Connect			: UA_Connect;
	SessionConnectInfo		: ST_UASessionConnectInfo;
	nConnectionHdl			: DWORD;
	(* Declarations for UA_GetNamespaceIndex *)
	fbUA_GetNamespaceIndex 	: UA_GetNamespaceIndex;
	nNamespaceIndex			: UINT;
	(* Declarations for UA_NodeGetHandle *)
	fbUA_NodeGetHandle		: UA_NodeGetHandle;
	NodeID					: ST_UANodeID;
	nNodeHdl				: DWORD;
	(* Declarations for UA_Read *)
	fbUA_Read				: UA_Read;
	stIndexRange			: ARRAY [1..nMaxIndexRange] OF ST_UAIndexRange;
	nIndexRangeCount		: UINT;
	stNodeAddInfo			: ST_UANodeAdditionalInfo;
	cbDataRead				: UDINT;
	(* Declarations for UA_NodeReleaseHandle *)
	fbUA_NodeReleaseHandle	: UA_NodeReleaseHandle;
	(* Declarations for UA_Disconnect *)
	fbUA_Disconnect			: UA_Disconnect;
END_VAR
VAR PERSISTENT
	sOpcUaServerUrl		: STRING(MAX_STRING_LENGTH) := 'opc.tcp://localhost:4840';
	sNamespaceUri		: STRING(MAX_STRING_LENGTH) := 'urn:BeckhoffAutomation:Ua:PLC1'; // TF6100 setup version 4.x default
END_VAR

CASE eState OF
	E_OPCUA_Client_Seq.Idle:
		IF (bExecute) THEN
			bError := FALSE;
			nErrorID := 0;
			bBusy := TRUE;
	
			SessionConnectInfo.tConnectTimeout := T#1M;
			SessionConnectInfo.tSessionTimeout := T#1M;
			SessionConnectInfo.sApplicationName := '';
			SessionConnectInfo.eSecurityMode := eUASecurityMsgMode_None;
			SessionConnectInfo.eSecurityPolicyUri := eUASecurityPolicy_None;
			SessionConnectInfo.eTransportProfileUri := eUATransportProfileUri_UATcp;
	
	(*		nIndexRange[1].nStartIndex := 0;
			nIndexRange[1].nEndIndex := 1;
			nIndexRange[1].bRangeAccess := TRUE; *)
			stNodeAddInfo.nIndexRangeCount := nIndexRangeCount;
			stNodeAddInfo.stIndexRange := stIndexRange;
			eState := E_OPCUA_Client_Seq.OpenSession;
		END_IF

	E_OPCUA_Client_Seq.CheckData:
		IF ((pTarget <> 0) AND (iTargetSize > 1)) THEN
			eState := E_OPCUA_Client_Seq.OpenSession;
		ELSE
			bError := TRUE;
			bBusy := FALSE;
			eState := E_OPCUA_Client_Seq.Done;
		END_IF

	E_OPCUA_Client_Seq.OpenSession:
		fbUA_Connect(	Execute := TRUE,
						ServerURL := sOpcUaServerUrl,
						SessionConnectInfo := SessionConnectInfo,
						Timeout := T#5S,
						ConnectionHdl => nConnectionHdl	);
	
		IF (NOT fbUA_Connect.Busy) THEN
			fbUA_Connect(Execute := FALSE);
			IF (NOT fbUA_Connect.Error) THEN
				// session opened
				eState := E_OPCUA_Client_Seq.GetNameSpace;
			ELSE
				bError := TRUE;
				nErrorID := fbUA_Connect.ErrorID;
				nConnectionHdl := 0;
				eState := E_OPCUA_Client_Seq.Idle;
			END_IF
		END_IF

	E_OPCUA_Client_Seq.GetNameSpace:
		fbUA_GetNamespaceIndex(	Execute := TRUE,
								ConnectionHdl := nConnectionHdl,
								NamespaceUri := sNamespaceUri,
								NamespaceIndex => nNamespaceIndex	);
	
		IF (NOT fbUA_GetNamespaceIndex.Busy) THEN
			fbUA_GetNamespaceIndex(Execute := FALSE);
			IF NOT fbUA_GetNamespaceIndex.Error THEN
				// Namespace index obtained
				eState := E_OPCUA_Client_Seq.GetNode;
			ELSE
				bError := TRUE;
				nErrorID := fbUA_GetNamespaceIndex.ErrorID;
				eState := E_OPCUA_Client_Seq.CloseSession;
			END_IF
		END_IF

	E_OPCUA_Client_Seq.GetNode:
		NodeID.eIdentifierType := eUAIdentifierType_String;
		NodeID.nNamespaceIndex := nNamespaceIndex;
		NodeID.sIdentifier := sVarName;
		fbUA_NodeGetHandle(	Execute := TRUE,
							ConnectionHdl := nConnectionHdl,
							NodeID := NodeID,
							NodeHdl => nNodeHdl	);
	
